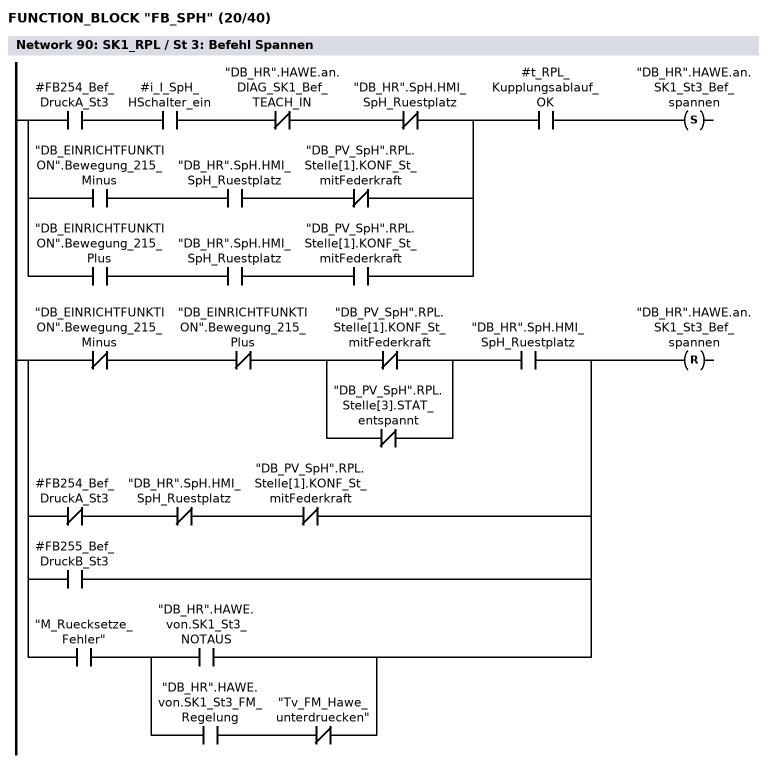

      U(    ;
      U     #FB254_Bef_DruckA_St3;
      U     #i_I_SpH_HSchalter_ein;
      UN    "DB_HR".HAWE.an.DIAG_SK1_Bef_TEACH_IN;
      UN    "DB_HR".SpH.HMI_SpH_Ruestplatz;
      O     ;
      U     "DB_EINRICHTFUNKTION".Bewegung_215_Minus;
      U     "DB_HR".SpH.HMI_SpH_Ruestplatz;
      UN    "DB_PV_SpH".RPL.Stelle[1].KONF_St_mitFederkraft;
      O     ;
      U     "DB_EINRICHTFUNKTION".Bewegung_215_Plus;
      U     "DB_HR".SpH.HMI_SpH_Ruestplatz;
      U     "DB_PV_SpH".RPL.Stelle[1].KONF_St_mitFederkraft;
      )     ;
      U     #t_RPL_Kupplungsablauf_OK;
      S     "DB_HR".HAWE.an.SK1_St3_Bef_spannen;

      U(    ;
      UN    "DB_EINRICHTFUNKTION".Bewegung_215_Minus;
      UN    "DB_EINRICHTFUNKTION".Bewegung_215_Plus;
      U(    ;
      ON    "DB_PV_SpH".RPL.Stelle[1].KONF_St_mitFederkraft;
      ON    "DB_PV_SpH".RPL.Stelle[3].STAT_entspannt;
      )     ;
      U     "DB_HR".SpH.HMI_SpH_Ruestplatz;
      O     ;
      UN    #FB254_Bef_DruckA_St3;
      UN    "DB_HR".SpH.HMI_SpH_Ruestplatz;
      UN    "DB_PV_SpH".RPL.Stelle[1].KONF_St_mitFederkraft;
      O     #FB255_Bef_DruckB_St3;
      O     ;
      U     "M_Ruecksetze_Fehler";
      U(    ;
      O     "DB_HR".HAWE.von.SK1_St3_NOTAUS;
      O     ;
      U     "DB_HR".HAWE.von.SK1_St3_FM_Regelung;
      UN    "Tv_FM_Hawe_unterdruecken";
      )     ;
      )     ;
      R     "DB_HR".HAWE.an.SK1_St3_Bef_spannen;
      NOP   0;
NETWORK
TITLE =SK1_RPL / St 4: Befehl Spannen
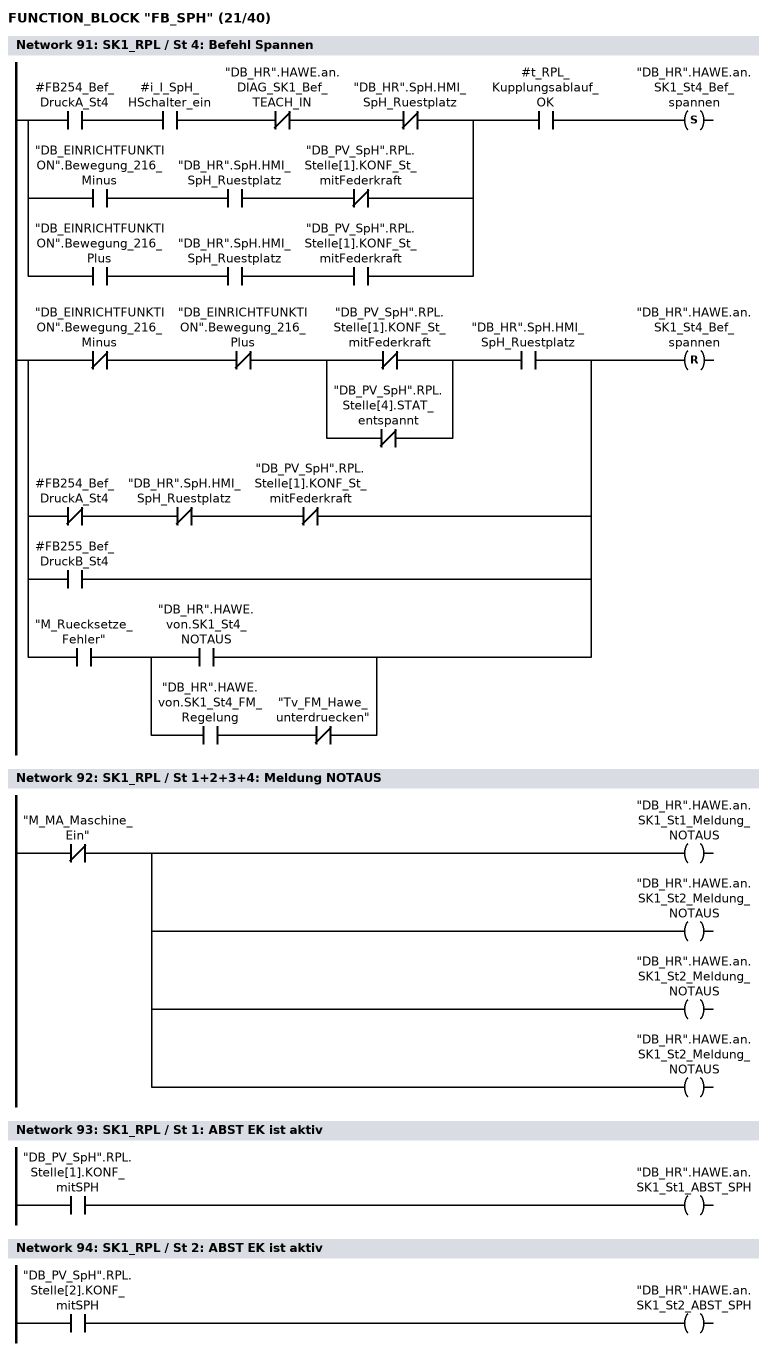

      U(    ;
      U     #FB254_Bef_DruckA_St4;
      U     #i_I_SpH_HSchalter_ein;
      UN    "DB_HR".HAWE.an.DIAG_SK1_Bef_TEACH_IN;
      UN    "DB_HR".SpH.HMI_SpH_Ruestplatz;
      O     ;
      U     "DB_EINRICHTFUNKTION".Bewegung_216_Minus;
      U     "DB_HR".SpH.HMI_SpH_Ruestplatz;
      UN    "DB_PV_SpH".RPL.Stelle[1].KONF_St_mitFederkraft;
      O     ;
      U     "DB_EINRICHTFUNKTION".Bewegung_216_Plus;
      U     "DB_HR".SpH.HMI_SpH_Ruestplatz;
      U     "DB_PV_SpH".RPL.Stelle[1].KONF_St_mitFederkraft;
      )     ;
      U     #t_RPL_Kupplungsablauf_OK;
      S     "DB_HR".HAWE.an.SK1_St4_Bef_spannen;

      U(    ;
      UN    "DB_EINRICHTFUNKTION".Bewegung_216_Minus;
      UN    "DB_EINRICHTFUNKTION".Bewegung_216_Plus;
      U(    ;
      ON    "DB_PV_SpH".RPL.Stelle[1].KONF_St_mitFederkraft;
      ON    "DB_PV_SpH".RPL.Stelle[4].STAT_entspannt;
      )     ;
      U     "DB_HR".SpH.HMI_SpH_Ruestplatz;
      O     ;
      UN    #FB254_Bef_DruckA_St4;
      UN    "DB_HR".SpH.HMI_SpH_Ruestplatz;
      UN    "DB_PV_SpH".RPL.Stelle[1].KONF_St_mitFederkraft;
      O     #FB255_Bef_DruckB_St4;
      O     ;
      U     "M_Ruecksetze_Fehler";
      U(    ;
      O     "DB_HR".HAWE.von.SK1_St4_NOTAUS;
      O     ;
      U     "DB_HR".HAWE.von.SK1_St4_FM_Regelung;
      UN    "Tv_FM_Hawe_unterdruecken";
      )     ;
      )     ;
      R     "DB_HR".HAWE.an.SK1_St4_Bef_spannen;
      NOP   0;
NETWORK
TITLE =SK1_RPL / St 1+2+3+4: Meldung NOTAUS

      UN    "M_MA_Maschine_Ein";
      =     "DB_HR".HAWE.an.SK1_St1_Meldung_NOTAUS;
      =     "DB_HR".HAWE.an.SK1_St2_Meldung_NOTAUS;
      =     "DB_HR".HAWE.an.SK1_St2_Meldung_NOTAUS;
      =     "DB_HR".HAWE.an.SK1_St2_Meldung_NOTAUS;
NETWORK
TITLE =SK1_RPL / St 1: ABST EK ist aktiv

      U     "DB_PV_SpH".RPL.Stelle[1].KONF_mitSPH;
      =     "DB_HR".HAWE.an.SK1_St1_ABST_SPH;
NETWORK
TITLE =SK1_RPL / St 2: ABST EK ist aktiv

      U     "DB_PV_SpH".RPL.Stelle[2].KONF_mitSPH;
      =     "DB_HR".HAWE.an.SK1_St2_ABST_SPH;
NETWORK
TITLE =SK1_RPL / St 3: ABST EK ist aktiv
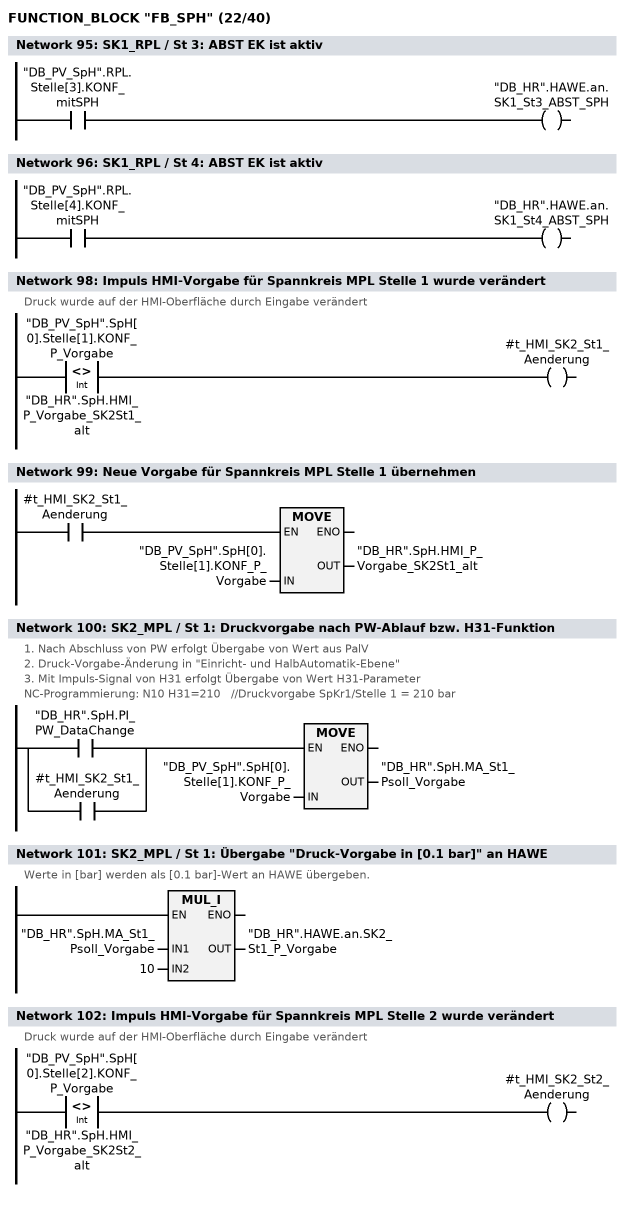

      U     "DB_PV_SpH".RPL.Stelle[3].KONF_mitSPH;
      =     "DB_HR".HAWE.an.SK1_St3_ABST_SPH;
NETWORK
TITLE =SK1_RPL / St 4: ABST EK ist aktiv

      U     "DB_PV_SpH".RPL.Stelle[4].KONF_mitSPH;
      =     "DB_HR".HAWE.an.SK1_St4_ABST_SPH;
NETWORK
TITLE =-------------- Maschinenplatz-Datenübergabe an HAWE ------------



NETWORK
TITLE =Impuls HMI-Vorgabe für Spannkreis MPL Stelle 1 wurde verändert
//Druck wurde auf der HMI-Oberfläche durch Eingabe verändert
      L     "DB_PV_SpH".SpH[0].Stelle[1].KONF_P_Vorgabe;
      L     "DB_HR".SpH.HMI_P_Vorgabe_SK2St1_alt;
      <>I   ;
      =     #t_HMI_SK2_St1_Aenderung;
NETWORK
TITLE =Neue Vorgabe für Spannkreis MPL Stelle 1 übernehmen

      U     #t_HMI_SK2_St1_Aenderung;
      SPBNB _00a;
      L     "DB_PV_SpH".SpH[0].Stelle[1].KONF_P_Vorgabe;
      T     "DB_HR".SpH.HMI_P_Vorgabe_SK2St1_alt;
_00a: NOP   0;
NETWORK
TITLE =SK2_MPL / St 1: Druckvorgabe nach PW-Ablauf bzw. H31-Funktion
//1. Nach Abschluss von PW erfolgt Übergabe von Wert aus PalV
//2. Druck-Vorgabe-Änderung in "Einricht- und HalbAutomatik-Ebene"
//3. Mit Impuls-Signal von H31 erfolgt Übergabe von Wert H31-Parameter
//   NC-Programmierung: N10 H31=210   //Druckvorgabe SpKr1/Stelle 1 = 210 bar
      U(    ;
      O     "DB_HR".SpH.PI_PW_DataChange;
      O     #t_HMI_SK2_St1_Aenderung;
      )     ;
      SPBNB _00b;
      L     "DB_PV_SpH".SpH[0].Stelle[1].KONF_P_Vorgabe;
      T     "DB_HR".SpH.MA_St1_Psoll_Vorgabe;
_00b: NOP   0;
NETWORK
TITLE =SK2_MPL / St 1: Übergabe "Druck-Vorgabe in [0.1 bar]" an HAWE
//Werte in [bar] werden als [0.1 bar]-Wert an HAWE übergeben.
      L     "DB_HR".SpH.MA_St1_Psoll_Vorgabe;
      L     10;
      *I    ;
      T     "DB_HR".HAWE.an.SK2_St1_P_Vorgabe;
NETWORK
TITLE =Impuls HMI-Vorgabe für Spannkreis MPL Stelle 2 wurde verändert
//Druck wurde auf der HMI-Oberfläche durch Eingabe verändert
      L     "DB_PV_SpH".SpH[0].Stelle[2].KONF_P_Vorgabe;
      L     "DB_HR".SpH.HMI_P_Vorgabe_SK2St2_alt;
      <>I   ;
      =     #t_HMI_SK2_St2_Aenderung;
NETWORK
TITLE =Neue Vorgabe für Spannkreis MPL Stelle 2 übernehmen
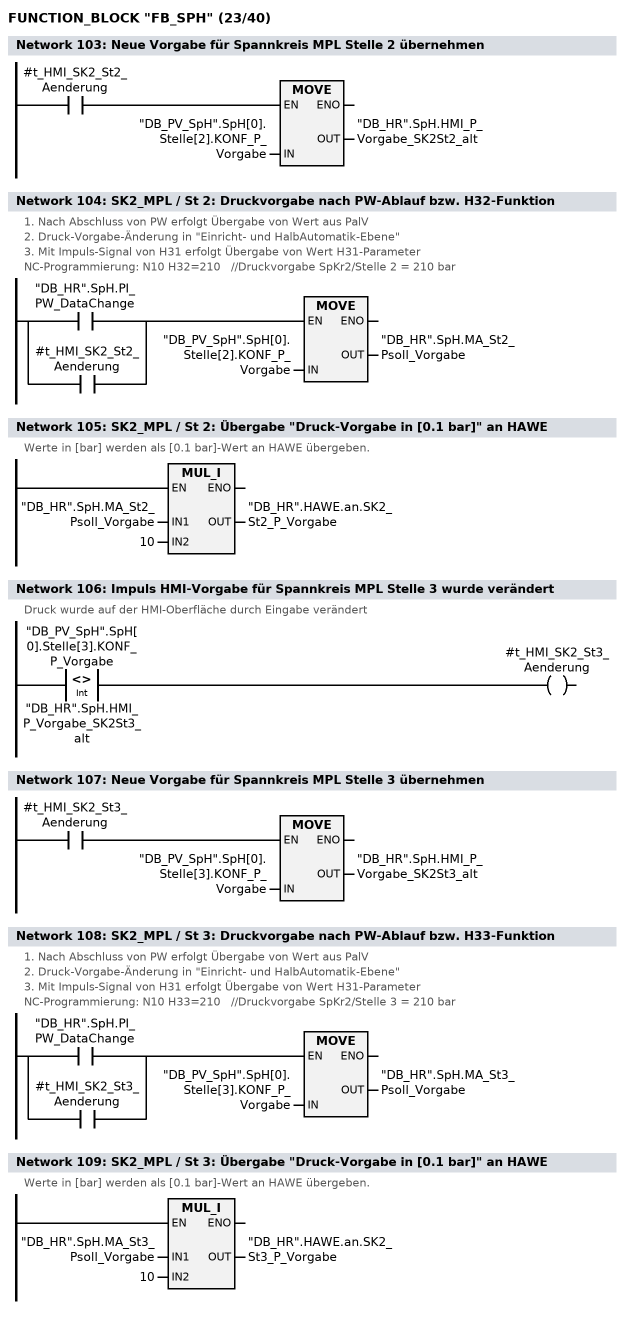

      U     #t_HMI_SK2_St2_Aenderung;
      SPBNB _00c;
      L     "DB_PV_SpH".SpH[0].Stelle[2].KONF_P_Vorgabe;
      T     "DB_HR".SpH.HMI_P_Vorgabe_SK2St2_alt;
_00c: NOP   0;
NETWORK
TITLE =SK2_MPL / St 2: Druckvorgabe nach PW-Ablauf bzw. H32-Funktion
//1. Nach Abschluss von PW erfolgt Übergabe von Wert aus PalV
//2. Druck-Vorgabe-Änderung in "Einricht- und HalbAutomatik-Ebene"
//3. Mit Impuls-Signal von H31 erfolgt Übergabe von Wert H31-Parameter
//   NC-Programmierung: N10 H32=210   //Druckvorgabe SpKr2/Stelle 2 = 210 bar
      U(    ;
      O     "DB_HR".SpH.PI_PW_DataChange;
      O     #t_HMI_SK2_St2_Aenderung;
      )     ;
      SPBNB _00d;
      L     "DB_PV_SpH".SpH[0].Stelle[2].KONF_P_Vorgabe;
      T     "DB_HR".SpH.MA_St2_Psoll_Vorgabe;
_00d: NOP   0;
NETWORK
TITLE =SK2_MPL / St 2: Übergabe "Druck-Vorgabe in [0.1 bar]" an HAWE
//Werte in [bar] werden als [0.1 bar]-Wert an HAWE übergeben.
      L     "DB_HR".SpH.MA_St2_Psoll_Vorgabe;
      L     10;
      *I    ;
      T     "DB_HR".HAWE.an.SK2_St2_P_Vorgabe;
NETWORK
TITLE =Impuls HMI-Vorgabe für Spannkreis MPL Stelle 3 wurde verändert
//Druck wurde auf der HMI-Oberfläche durch Eingabe verändert
      L     "DB_PV_SpH".SpH[0].Stelle[3].KONF_P_Vorgabe;
      L     "DB_HR".SpH.HMI_P_Vorgabe_SK2St3_alt;
      <>I   ;
      =     #t_HMI_SK2_St3_Aenderung;
NETWORK
TITLE =Neue Vorgabe für Spannkreis MPL Stelle 3 übernehmen

      U     #t_HMI_SK2_St3_Aenderung;
      SPBNB _00e;
      L     "DB_PV_SpH".SpH[0].Stelle[3].KONF_P_Vorgabe;
      T     "DB_HR".SpH.HMI_P_Vorgabe_SK2St3_alt;
_00e: NOP   0;
NETWORK
TITLE =SK2_MPL / St 3: Druckvorgabe nach PW-Ablauf bzw. H33-Funktion
//1. Nach Abschluss von PW erfolgt Übergabe von Wert aus PalV
//2. Druck-Vorgabe-Änderung in "Einricht- und HalbAutomatik-Ebene"
//3. Mit Impuls-Signal von H31 erfolgt Übergabe von Wert H31-Parameter
//   NC-Programmierung: N10 H33=210   //Druckvorgabe SpKr2/Stelle 3 = 210 bar
      U(    ;
      O     "DB_HR".SpH.PI_PW_DataChange;
      O     #t_HMI_SK2_St3_Aenderung;
      )     ;
      SPBNB _00f;
      L     "DB_PV_SpH".SpH[0].Stelle[3].KONF_P_Vorgabe;
      T     "DB_HR".SpH.MA_St3_Psoll_Vorgabe;
_00f: NOP   0;
NETWORK
TITLE =SK2_MPL / St 3: Übergabe "Druck-Vorgabe in [0.1 bar]" an HAWE
//Werte in [bar] werden als [0.1 bar]-Wert an HAWE übergeben.
      L     "DB_HR".SpH.MA_St3_Psoll_Vorgabe;
      L     10;
      *I    ;
      T     "DB_HR".HAWE.an.SK2_St3_P_Vorgabe;
NETWORK
TITLE =Impuls HMI-Vorgabe für Spannkreis MPL Stelle 4 wurde verändert
//Druck wurde auf der HMI-Oberfläche durch Eingabe verändert
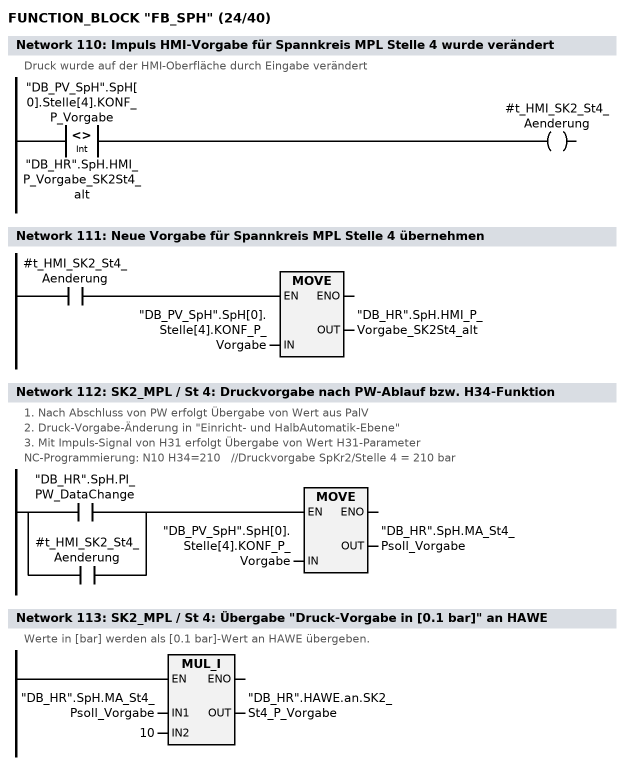
      L     "DB_PV_SpH".SpH[0].Stelle[4].KONF_P_Vorgabe;
      L     "DB_HR".SpH.HMI_P_Vorgabe_SK2St4_alt;
      <>I   ;
      =     #t_HMI_SK2_St4_Aenderung;
NETWORK
TITLE =Neue Vorgabe für Spannkreis MPL Stelle 4 übernehmen

      U     #t_HMI_SK2_St4_Aenderung;
      SPBNB _010;
      L     "DB_PV_SpH".SpH[0].Stelle[4].KONF_P_Vorgabe;
      T     "DB_HR".SpH.HMI_P_Vorgabe_SK2St4_alt;
_010: NOP   0;
NETWORK
TITLE =SK2_MPL / St 4: Druckvorgabe nach PW-Ablauf bzw. H34-Funktion
//1. Nach Abschluss von PW erfolgt Übergabe von Wert aus PalV
//2. Druck-Vorgabe-Änderung in "Einricht- und HalbAutomatik-Ebene"
//3. Mit Impuls-Signal von H31 erfolgt Übergabe von Wert H31-Parameter
//   NC-Programmierung: N10 H34=210   //Druckvorgabe SpKr2/Stelle 4 = 210 bar
      U(    ;
      O     "DB_HR".SpH.PI_PW_DataChange;
      O     #t_HMI_SK2_St4_Aenderung;
      )     ;
      SPBNB _011;
      L     "DB_PV_SpH".SpH[0].Stelle[4].KONF_P_Vorgabe;
      T     "DB_HR".SpH.MA_St4_Psoll_Vorgabe;
_011: NOP   0;
NETWORK
TITLE =SK2_MPL / St 4: Übergabe "Druck-Vorgabe in [0.1 bar]" an HAWE
//Werte in [bar] werden als [0.1 bar]-Wert an HAWE übergeben.
      L     "DB_HR".SpH.MA_St4_Psoll_Vorgabe;
      L     10;
      *I    ;
      T     "DB_HR".HAWE.an.SK2_St4_P_Vorgabe;
NETWORK
TITLE =H31-Funktion
//i_REAL_H_wert           := REAL-Wert der H-Funktion
//i_T_Ausgang_Entspannen  := Timer-Ausgang: Spannstelle entspannen
//i_HAWE_Druck_erreicht   := Meldung von HAWE "Druck erreicht"
//i_RESET_offene_Stelle_OK:= RESET Funktion "offene Spannstelle"
//                           z.B. PW-Ablauf aktiv
//i_Spannstelle_aktiv     := Spannstelle konfiguriert
//o_HFKT_quitpflichtig    := Merker für H-Funktion "Quittierungspflichtig"
//o_HFKT_Quittung         := Merker für H-Funktion "Quittierung"
//o_FM_falscher_Wert      := FM "Falscher Wert bei H-Eingabe"
//o_T_Start_Entspannen    := Timer-Start: Spannstelle entspannen
//o_T_Vorgabe_Entspannen  := Timer-Vorgabe: Spannstelle entspannen [s]
//o_kein_OVR_ist_0        := kein OVR=0 aktivieren
//                           a) Überwachung ist ausgeschaltet
//                           b) Spannstelle wurde geöffnet
//io_akt_Druckvorgabe     := Aktuelle Druckvorgabe (Sollwert in Maschine)
//io_M_H_FKT              := Merker für H-Funktion aktiv
//io_Bef_Entspannen       := Befehl an Hawe "Spannstelle entspannen"
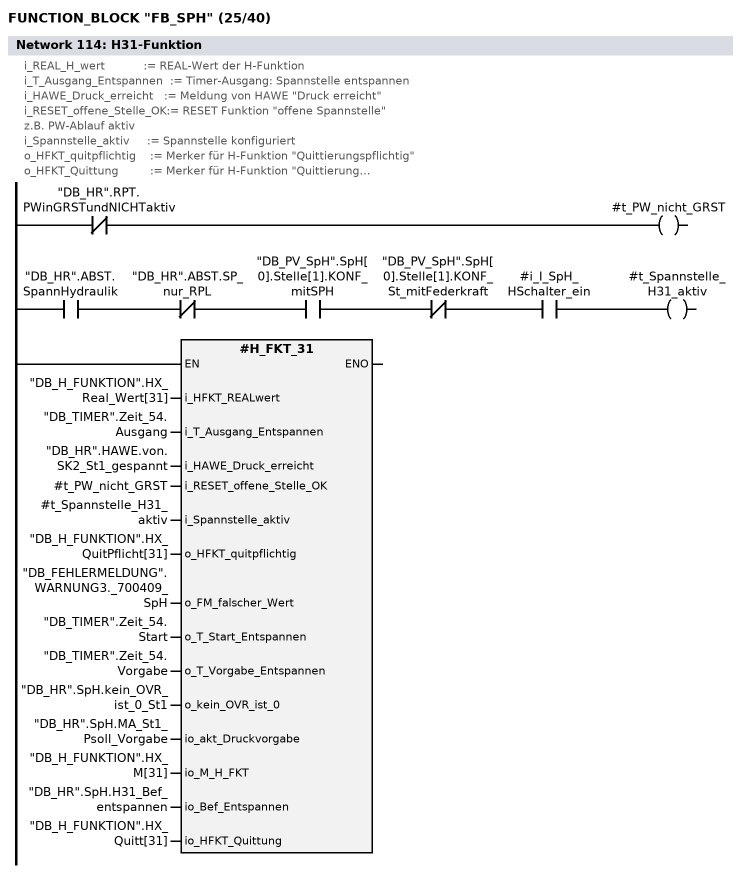
      UN    "DB_HR".RPT.PWinGRSTundNICHTaktiv;
      =     #t_PW_nicht_GRST;

      U     "DB_HR".ABST.SpannHydraulik;
      UN    "DB_HR".ABST.SP_nur_RPL;
      U     "DB_PV_SpH".SpH[0].Stelle[1].KONF_mitSPH;
      UN    "DB_PV_SpH".SpH[0].Stelle[1].KONF_St_mitFederkraft;
      U     #i_I_SpH_HSchalter_ein;
      =     #t_Spannstelle_H31_aktiv;

      CALL #H_FKT_31 (
           i_HFKT_REALwert          := "DB_H_FUNKTION".HX_Real_Wert[31],
           i_T_Ausgang_Entspannen   := "DB_TIMER".Zeit_54.Ausgang,
           i_HAWE_Druck_erreicht    := "DB_HR".HAWE.von.SK2_St1_gespannt,
           i_RESET_offene_Stelle_OK := #t_PW_nicht_GRST,
           i_Spannstelle_aktiv      := #t_Spannstelle_H31_aktiv,
           o_HFKT_quitpflichtig     := "DB_H_FUNKTION".HX_QuitPflicht[31],
           o_FM_falscher_Wert       := "DB_FEHLERMELDUNG".WARNUNG3._700409_SpH,
           o_T_Start_Entspannen     := "DB_TIMER".Zeit_54.Start,
           o_T_Vorgabe_Entspannen   := "DB_TIMER".Zeit_54.Vorgabe,
           o_kein_OVR_ist_0         := "DB_HR".SpH.kein_OVR_ist_0_St1,
           io_akt_Druckvorgabe      := "DB_HR".SpH.MA_St1_Psoll_Vorgabe,
           io_M_H_FKT               := "DB_H_FUNKTION".HX_M[31],
           io_Bef_Entspannen        := "DB_HR".SpH.H31_Bef_entspannen,
           io_HFKT_Quittung         := "DB_H_FUNKTION".HX_Quitt[31]);

NETWORK
TITLE =H32-Funktion
//i_REAL_H_wert           := REAL-Wert der H-Funktion
//i_T_Ausgang_Entspannen  := Timer-Ausgang: Spannstelle entspannen
//i_HAWE_Druck_erreicht   := Meldung von HAWE "Druck erreicht"
//i_RESET_offene_Stelle_OK:= RESET Funktion "offene Spannstelle"
//                           z.B. PW-Ablauf aktiv
//i_Spannstelle_aktiv     := Spannstelle konfiguriert
//o_HFKT_quitpflichtig    := Merker für H-Funktion "Quittierungspflichtig"
//o_HFKT_Quittung         := Merker für H-Funktion "Quittierung"
//o_FM_falscher_Wert      := FM "Falscher Wert bei H-Eingabe"
//o_T_Start_Entspannen    := Timer-Start: Spannstelle entspannen
//o_T_Vorgabe_Entspannen  := Timer-Vorgabe: Spannstelle entspannen [s]
//o_kein_OVR_ist_0        := kein OVR=0 aktivieren
//                           a) Überwachung ist ausgeschaltet
//                           b) Spannstelle wurde geöffnet
//io_akt_Druckvorgabe     := Aktuelle Druckvorgabe (Sollwert in Maschine)
//io_M_H_FKT              := Merker für H-Funktion aktiv
//io_Bef_Entspannen       := Befehl an Hawe "Spannstelle entspannen"
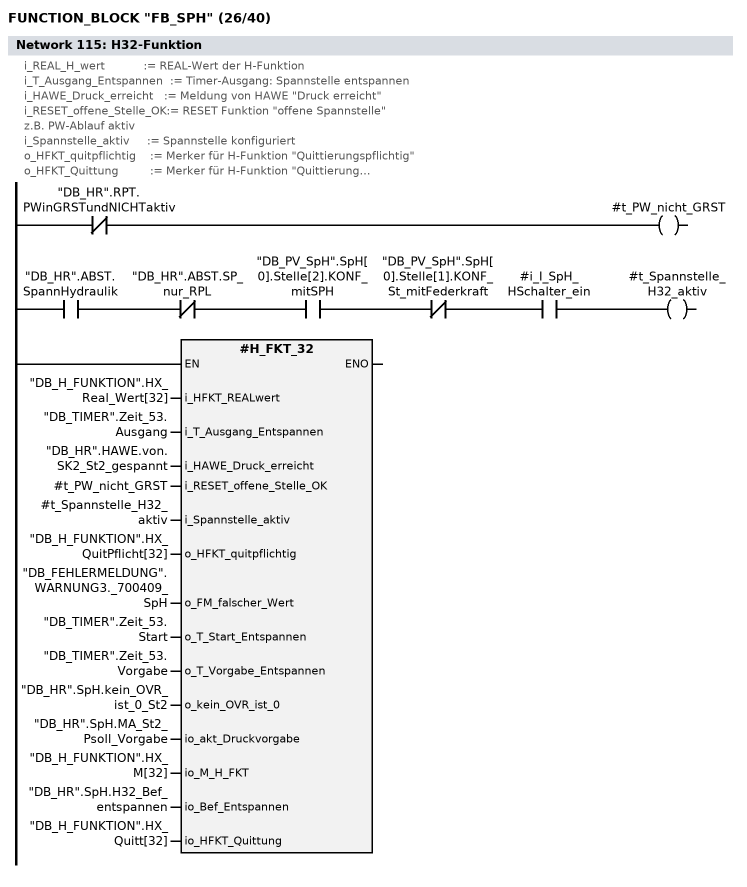
      UN    "DB_HR".RPT.PWinGRSTundNICHTaktiv;
      =     #t_PW_nicht_GRST;

      U     "DB_HR".ABST.SpannHydraulik;
      UN    "DB_HR".ABST.SP_nur_RPL;
      U     "DB_PV_SpH".SpH[0].Stelle[2].KONF_mitSPH;
      UN    "DB_PV_SpH".SpH[0].Stelle[1].KONF_St_mitFederkraft;
      U     #i_I_SpH_HSchalter_ein;
      =     #t_Spannstelle_H32_aktiv;

      CALL #H_FKT_32 (
           i_HFKT_REALwert          := "DB_H_FUNKTION".HX_Real_Wert[32],
           i_T_Ausgang_Entspannen   := "DB_TIMER".Zeit_53.Ausgang,
           i_HAWE_Druck_erreicht    := "DB_HR".HAWE.von.SK2_St2_gespannt,
           i_RESET_offene_Stelle_OK := #t_PW_nicht_GRST,
           i_Spannstelle_aktiv      := #t_Spannstelle_H32_aktiv,
           o_HFKT_quitpflichtig     := "DB_H_FUNKTION".HX_QuitPflicht[32],
           o_FM_falscher_Wert       := "DB_FEHLERMELDUNG".WARNUNG3._700409_SpH,
           o_T_Start_Entspannen     := "DB_TIMER".Zeit_53.Start,
           o_T_Vorgabe_Entspannen   := "DB_TIMER".Zeit_53.Vorgabe,
           o_kein_OVR_ist_0         := "DB_HR".SpH.kein_OVR_ist_0_St2,
           io_akt_Druckvorgabe      := "DB_HR".SpH.MA_St2_Psoll_Vorgabe,
           io_M_H_FKT               := "DB_H_FUNKTION".HX_M[32],
           io_Bef_Entspannen        := "DB_HR".SpH.H32_Bef_entspannen,
           io_HFKT_Quittung         := "DB_H_FUNKTION".HX_Quitt[32]);

NETWORK
TITLE =H33-Funktion
//i_REAL_H_wert           := REAL-Wert der H-Funktion
//i_T_Ausgang_Entspannen  := Timer-Ausgang: Spannstelle entspannen
//i_HAWE_Druck_erreicht   := Meldung von HAWE "Druck erreicht"
//i_RESET_offene_Stelle_OK:= RESET Funktion "offene Spannstelle"
//                           z.B. PW-Ablauf aktiv
//i_Spannstelle_aktiv     := Spannstelle konfiguriert
//o_HFKT_quitpflichtig    := Merker für H-Funktion "Quittierungspflichtig"
//o_HFKT_Quittung         := Merker für H-Funktion "Quittierung"
//o_FM_falscher_Wert      := FM "Falscher Wert bei H-Eingabe"
//o_T_Start_Entspannen    := Timer-Start: Spannstelle entspannen
//o_T_Vorgabe_Entspannen  := Timer-Vorgabe: Spannstelle entspannen [s]
//o_kein_OVR_ist_0        := kein OVR=0 aktivieren
//                           a) Überwachung ist ausgeschaltet
//                           b) Spannstelle wurde geöffnet
//io_akt_Druckvorgabe     := Aktuelle Druckvorgabe (Sollwert in Maschine)
//io_M_H_FKT              := Merker für H-Funktion aktiv
//io_Bef_Entspannen       := Befehl an Hawe "Spannstelle entspannen"
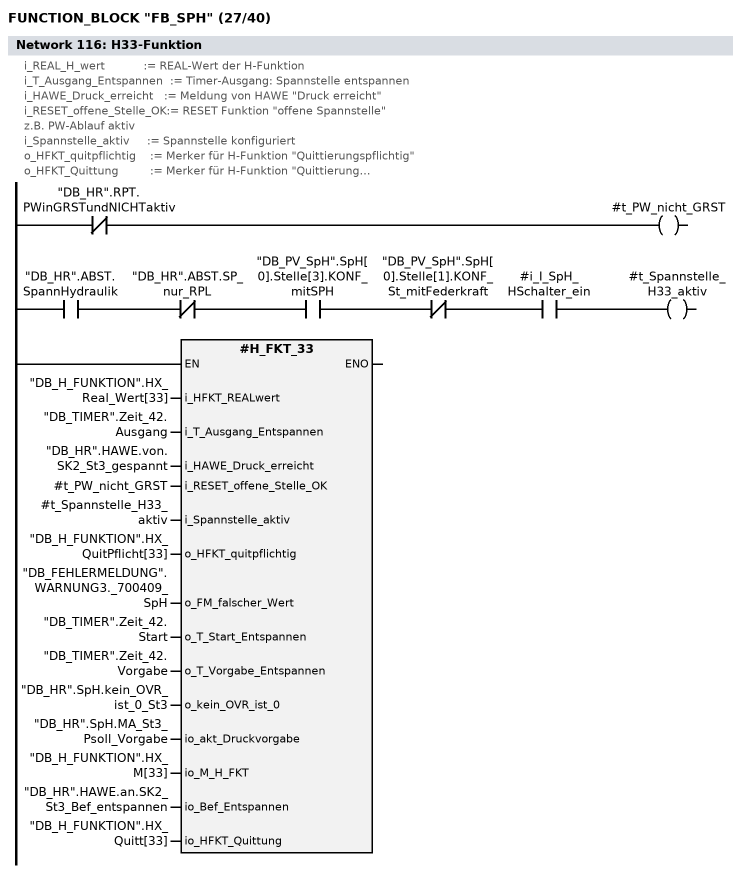
      UN    "DB_HR".RPT.PWinGRSTundNICHTaktiv;
      =     #t_PW_nicht_GRST;

      U     "DB_HR".ABST.SpannHydraulik;
      UN    "DB_HR".ABST.SP_nur_RPL;
      U     "DB_PV_SpH".SpH[0].Stelle[3].KONF_mitSPH;
      UN    "DB_PV_SpH".SpH[0].Stelle[1].KONF_St_mitFederkraft;
      U     #i_I_SpH_HSchalter_ein;
      =     #t_Spannstelle_H33_aktiv;


      CALL #H_FKT_33 (
           i_HFKT_REALwert          := "DB_H_FUNKTION".HX_Real_Wert[33],
           i_T_Ausgang_Entspannen   := "DB_TIMER".Zeit_42.Ausgang,
           i_HAWE_Druck_erreicht    := "DB_HR".HAWE.von.SK2_St3_gespannt,
           i_RESET_offene_Stelle_OK := #t_PW_nicht_GRST,
           i_Spannstelle_aktiv      := #t_Spannstelle_H33_aktiv,
           o_HFKT_quitpflichtig     := "DB_H_FUNKTION".HX_QuitPflicht[33],
           o_FM_falscher_Wert       := "DB_FEHLERMELDUNG".WARNUNG3._700409_SpH,
           o_T_Start_Entspannen     := "DB_TIMER".Zeit_42.Start,
           o_T_Vorgabe_Entspannen   := "DB_TIMER".Zeit_42.Vorgabe,
           o_kein_OVR_ist_0         := "DB_HR".SpH.kein_OVR_ist_0_St3,
           io_akt_Druckvorgabe      := "DB_HR".SpH.MA_St3_Psoll_Vorgabe,
           io_M_H_FKT               := "DB_H_FUNKTION".HX_M[33],
           io_Bef_Entspannen        := "DB_HR".HAWE.an.SK2_St3_Bef_entspannen,
           io_HFKT_Quittung         := "DB_H_FUNKTION".HX_Quitt[33]);

NETWORK
TITLE =H34-Funktion
//i_REAL_H_wert           := REAL-Wert der H-Funktion
//i_T_Ausgang_Entspannen  := Timer-Ausgang: Spannstelle entspannen
//i_HAWE_Druck_erreicht   := Meldung von HAWE "Druck erreicht"
//i_RESET_offene_Stelle_OK:= RESET Funktion "offene Spannstelle"
//                           z.B. PW-Ablauf aktiv
//i_Spannstelle_aktiv     := Spannstelle konfiguriert
//o_HFKT_quitpflichtig    := Merker für H-Funktion "Quittierungspflichtig"
//o_HFKT_Quittung         := Merker für H-Funktion "Quittierung"
//o_FM_falscher_Wert      := FM "Falscher Wert bei H-Eingabe"
//o_T_Start_Entspannen    := Timer-Start: Spannstelle entspannen
//o_T_Vorgabe_Entspannen  := Timer-Vorgabe: Spannstelle entspannen [s]
//o_kein_OVR_ist_0        := kein OVR=0 aktivieren
//                           a) Überwachung ist ausgeschaltet
//                           b) Spannstelle wurde geöffnet
//io_akt_Druckvorgabe     := Aktuelle Druckvorgabe (Sollwert in Maschine)
//io_M_H_FKT              := Merker für H-Funktion aktiv
//io_Bef_Entspannen       := Befehl an Hawe "Spannstelle entspannen"
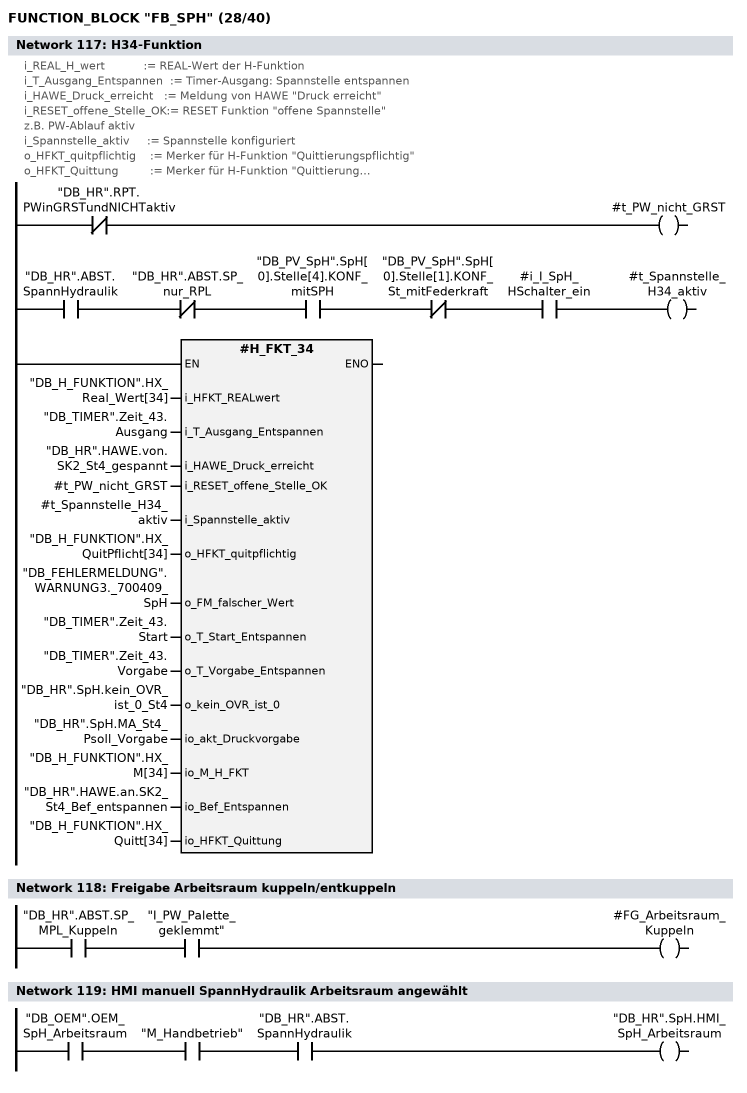
      UN    "DB_HR".RPT.PWinGRSTundNICHTaktiv;
      =     #t_PW_nicht_GRST;

      U     "DB_HR".ABST.SpannHydraulik;
      UN    "DB_HR".ABST.SP_nur_RPL;
      U     "DB_PV_SpH".SpH[0].Stelle[4].KONF_mitSPH;
      UN    "DB_PV_SpH".SpH[0].Stelle[1].KONF_St_mitFederkraft;
      U     #i_I_SpH_HSchalter_ein;
      =     #t_Spannstelle_H34_aktiv;

      CALL #H_FKT_34 (
           i_HFKT_REALwert          := "DB_H_FUNKTION".HX_Real_Wert[34],
           i_T_Ausgang_Entspannen   := "DB_TIMER".Zeit_43.Ausgang,
           i_HAWE_Druck_erreicht    := "DB_HR".HAWE.von.SK2_St4_gespannt,
           i_RESET_offene_Stelle_OK := #t_PW_nicht_GRST,
           i_Spannstelle_aktiv      := #t_Spannstelle_H34_aktiv,
           o_HFKT_quitpflichtig     := "DB_H_FUNKTION".HX_QuitPflicht[34],
           o_FM_falscher_Wert       := "DB_FEHLERMELDUNG".WARNUNG3._700409_SpH,
           o_T_Start_Entspannen     := "DB_TIMER".Zeit_43.Start,
           o_T_Vorgabe_Entspannen   := "DB_TIMER".Zeit_43.Vorgabe,
           o_kein_OVR_ist_0         := "DB_HR".SpH.kein_OVR_ist_0_St4,
           io_akt_Druckvorgabe      := "DB_HR".SpH.MA_St4_Psoll_Vorgabe,
           io_M_H_FKT               := "DB_H_FUNKTION".HX_M[34],
           io_Bef_Entspannen        := "DB_HR".HAWE.an.SK2_St4_Bef_entspannen,
           io_HFKT_Quittung         := "DB_H_FUNKTION".HX_Quitt[34]);
NETWORK
TITLE =Freigabe Arbeitsraum kuppeln/entkuppeln

      U     "DB_HR".ABST.SP_MPL_Kuppeln;
      U     "I_PW_Palette_geklemmt";
      =     #FG_Arbeitsraum_Kuppeln;
NETWORK
TITLE =HMI manuell SpannHydraulik Arbeitsraum angewählt

      U     "DB_OEM".OEM_SpH_Arbeitsraum;
      U     "M_Handbetrieb";
      U     "DB_HR".ABST.SpannHydraulik;
      =     "DB_HR".SpH.HMI_SpH_Arbeitsraum;
NETWORK
TITLE =HMI-Manuell: Maschinenraum Stelle 1
//HMI: Manuell / [SK5] Hand-Fkt SpannHydr.   Bild-Nr: 37
//                                           Bewegungs-Nr: 219
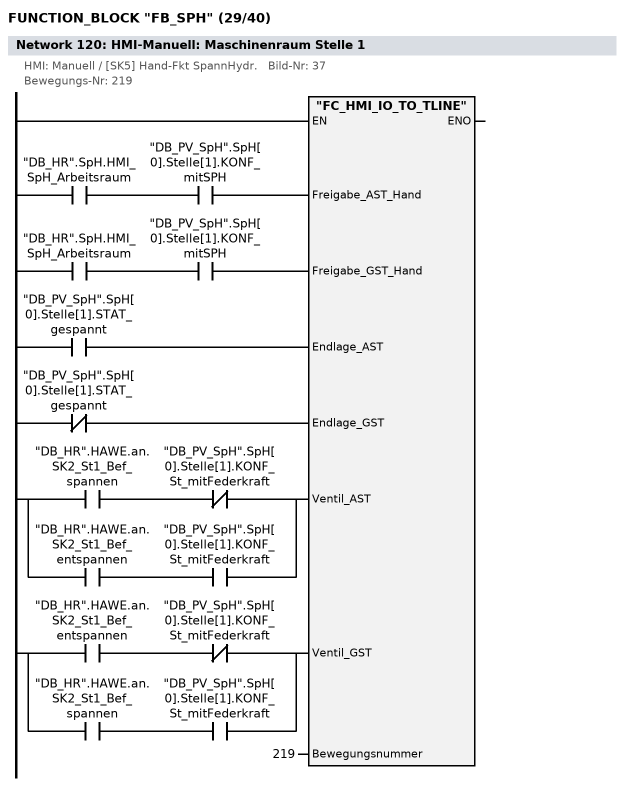
      U     "DB_HR".SpH.HMI_SpH_Arbeitsraum;
      U     "DB_PV_SpH".SpH[0].Stelle[1].KONF_mitSPH;
      =     L     18.0;
      BLD   103;
      U     "DB_HR".SpH.HMI_SpH_Arbeitsraum;
      U     "DB_PV_SpH".SpH[0].Stelle[1].KONF_mitSPH;
      =     L     18.1;
      BLD   103;
      U     "DB_PV_SpH".SpH[0].Stelle[1].STAT_gespannt;
      =     L     18.2;
      BLD   103;
      UN    "DB_PV_SpH".SpH[0].Stelle[1].STAT_gespannt;
      =     L     18.3;
      BLD   103;
      U(    ;
      U     "DB_HR".HAWE.an.SK2_St1_Bef_spannen;
      UN    "DB_PV_SpH".SpH[0].Stelle[1].KONF_St_mitFederkraft;
      O     ;
      U     "DB_HR".HAWE.an.SK2_St1_Bef_entspannen;
      U     "DB_PV_SpH".SpH[0].Stelle[1].KONF_St_mitFederkraft;
      )     ;
      =     L     18.4;
      BLD   103;
      U(    ;
      U     "DB_HR".HAWE.an.SK2_St1_Bef_entspannen;
      UN    "DB_PV_SpH".SpH[0].Stelle[1].KONF_St_mitFederkraft;
      O     ;
      U     "DB_HR".HAWE.an.SK2_St1_Bef_spannen;
      U     "DB_PV_SpH".SpH[0].Stelle[1].KONF_St_mitFederkraft;
      )     ;
      =     L     18.5;
      BLD   103;
      CALL "FC_HMI_IO_TO_TLINE" (
           Freigabe_AST_Hand        := L     18.0,
           Freigabe_GST_Hand        := L     18.1,
           Endlage_AST              := L     18.2,
           Endlage_GST              := L     18.3,
           Ventil_AST               := L     18.4,
           Ventil_GST               := L     18.5,
           Bewegungsnummer          := 219);
      NOP   0;
NETWORK
TITLE =HMI-Manuell: Maschinenraum Stelle 2
//HMI: Manuell / [SK5] Hand-Fkt SpannHydr.   Bild-Nr: 37
//                                           Bewegungs-Nr: 220
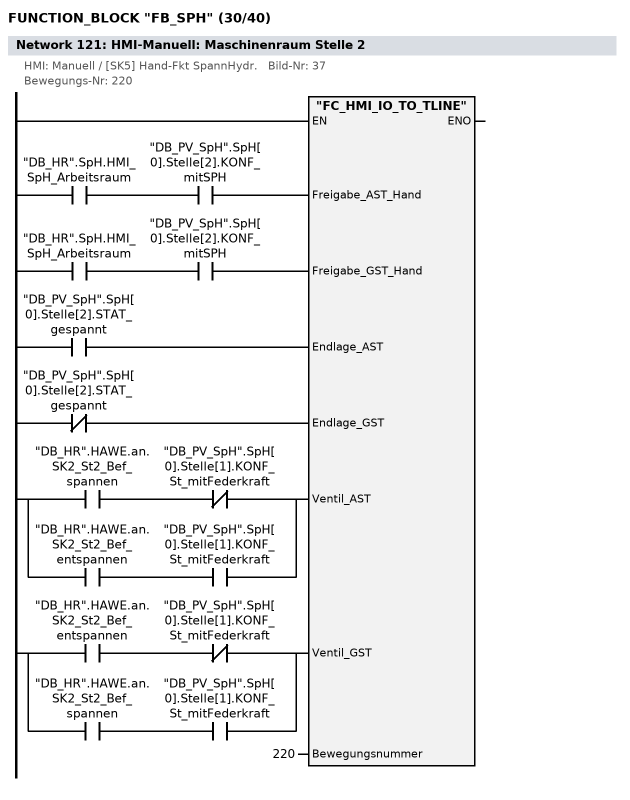
      U     "DB_HR".SpH.HMI_SpH_Arbeitsraum;
      U     "DB_PV_SpH".SpH[0].Stelle[2].KONF_mitSPH;
      =     L     18.0;
      BLD   103;
      U     "DB_HR".SpH.HMI_SpH_Arbeitsraum;
      U     "DB_PV_SpH".SpH[0].Stelle[2].KONF_mitSPH;
      =     L     18.1;
      BLD   103;
      U     "DB_PV_SpH".SpH[0].Stelle[2].STAT_gespannt;
      =     L     18.2;
      BLD   103;
      UN    "DB_PV_SpH".SpH[0].Stelle[2].STAT_gespannt;
      =     L     18.3;
      BLD   103;
      U(    ;
      U     "DB_HR".HAWE.an.SK2_St2_Bef_spannen;
      UN    "DB_PV_SpH".SpH[0].Stelle[1].KONF_St_mitFederkraft;
      O     ;
      U     "DB_HR".HAWE.an.SK2_St2_Bef_entspannen;
      U     "DB_PV_SpH".SpH[0].Stelle[1].KONF_St_mitFederkraft;
      )     ;
      =     L     18.4;
      BLD   103;
      U(    ;
      U     "DB_HR".HAWE.an.SK2_St2_Bef_entspannen;
      UN    "DB_PV_SpH".SpH[0].Stelle[1].KONF_St_mitFederkraft;
      O     ;
      U     "DB_HR".HAWE.an.SK2_St2_Bef_spannen;
      U     "DB_PV_SpH".SpH[0].Stelle[1].KONF_St_mitFederkraft;
      )     ;
      =     L     18.5;
      BLD   103;
      CALL "FC_HMI_IO_TO_TLINE" (
           Freigabe_AST_Hand        := L     18.0,
           Freigabe_GST_Hand        := L     18.1,
           Endlage_AST              := L     18.2,
           Endlage_GST              := L     18.3,
           Ventil_AST               := L     18.4,
           Ventil_GST               := L     18.5,
           Bewegungsnummer          := 220);
      NOP   0;
NETWORK
TITLE =HMI-Manuell: Maschinenraum Stelle 3
//HMI: Manuell / [SK5] Hand-Fkt SpannHydr.   Bild-Nr: 37
//                                           Bewegungs-Nr: 221
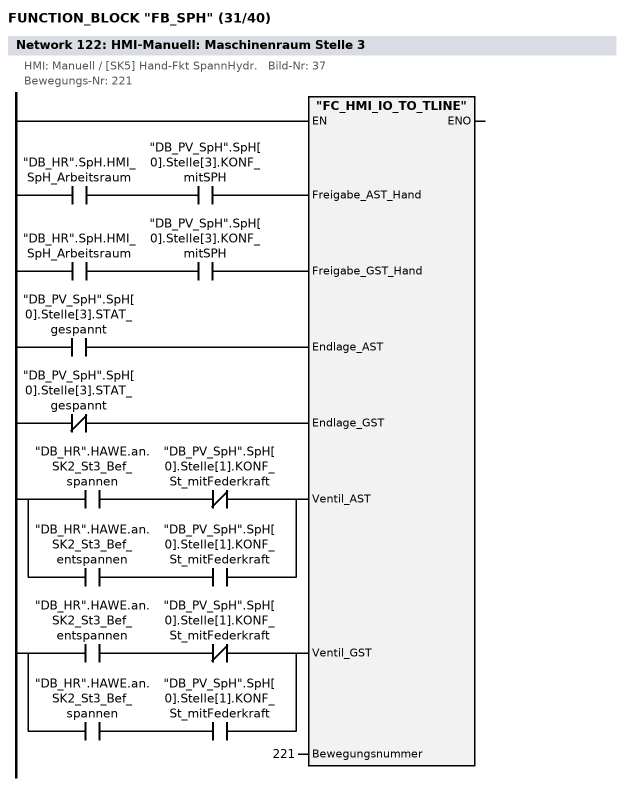
      U     "DB_HR".SpH.HMI_SpH_Arbeitsraum;
      U     "DB_PV_SpH".SpH[0].Stelle[3].KONF_mitSPH;
      =     L     18.0;
      BLD   103;
      U     "DB_HR".SpH.HMI_SpH_Arbeitsraum;
      U     "DB_PV_SpH".SpH[0].Stelle[3].KONF_mitSPH;
      =     L     18.1;
      BLD   103;
      U     "DB_PV_SpH".SpH[0].Stelle[3].STAT_gespannt;
      =     L     18.2;
      BLD   103;
      UN    "DB_PV_SpH".SpH[0].Stelle[3].STAT_gespannt;
      =     L     18.3;
      BLD   103;
      U(    ;
      U     "DB_HR".HAWE.an.SK2_St3_Bef_spannen;
      UN    "DB_PV_SpH".SpH[0].Stelle[1].KONF_St_mitFederkraft;
      O     ;
      U     "DB_HR".HAWE.an.SK2_St3_Bef_entspannen;
      U     "DB_PV_SpH".SpH[0].Stelle[1].KONF_St_mitFederkraft;
      )     ;
      =     L     18.4;
      BLD   103;
      U(    ;
      U     "DB_HR".HAWE.an.SK2_St3_Bef_entspannen;
      UN    "DB_PV_SpH".SpH[0].Stelle[1].KONF_St_mitFederkraft;
      O     ;
      U     "DB_HR".HAWE.an.SK2_St3_Bef_spannen;
      U     "DB_PV_SpH".SpH[0].Stelle[1].KONF_St_mitFederkraft;
      )     ;
      =     L     18.5;
      BLD   103;
      CALL "FC_HMI_IO_TO_TLINE" (
           Freigabe_AST_Hand        := L     18.0,
           Freigabe_GST_Hand        := L     18.1,
           Endlage_AST              := L     18.2,
           Endlage_GST              := L     18.3,
           Ventil_AST               := L     18.4,
           Ventil_GST               := L     18.5,
           Bewegungsnummer          := 221);
      NOP   0;
NETWORK
TITLE =HMI-Manuell: Maschinenraum Stelle 4
//HMI: Manuell / [SK5] Hand-Fkt SpannHydr.   Bild-Nr: 37
//                                           Bewegungs-Nr: 222
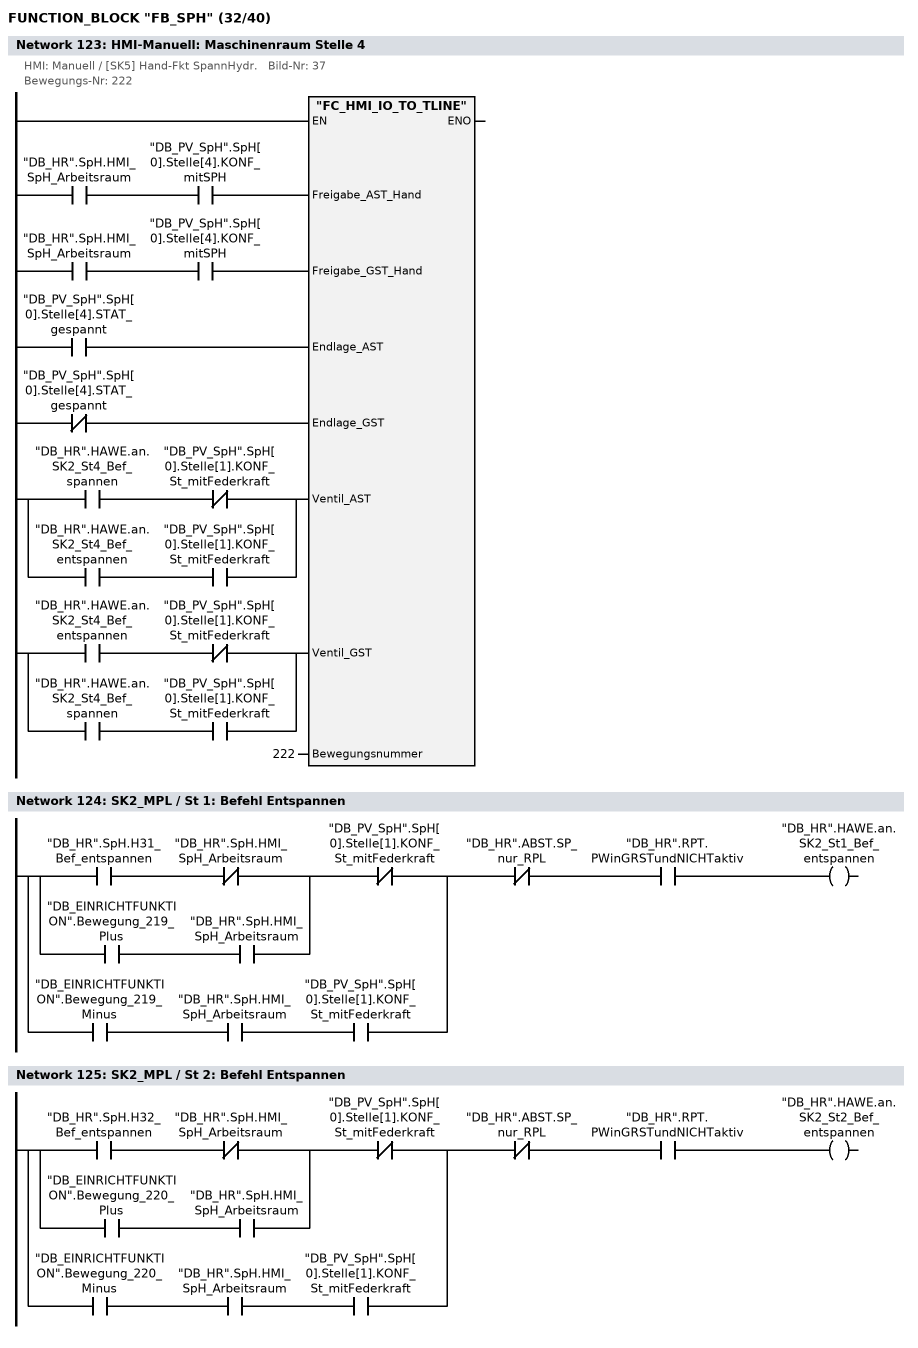
      U     "DB_HR".SpH.HMI_SpH_Arbeitsraum;
      U     "DB_PV_SpH".SpH[0].Stelle[4].KONF_mitSPH;
      =     L     18.0;
      BLD   103;
      U     "DB_HR".SpH.HMI_SpH_Arbeitsraum;
      U     "DB_PV_SpH".SpH[0].Stelle[4].KONF_mitSPH;
      =     L     18.1;
      BLD   103;
      U     "DB_PV_SpH".SpH[0].Stelle[4].STAT_gespannt;
      =     L     18.2;
      BLD   103;
      UN    "DB_PV_SpH".SpH[0].Stelle[4].STAT_gespannt;
      =     L     18.3;
      BLD   103;
      U(    ;
      U     "DB_HR".HAWE.an.SK2_St4_Bef_spannen;
      UN    "DB_PV_SpH".SpH[0].Stelle[1].KONF_St_mitFederkraft;
      O     ;
      U     "DB_HR".HAWE.an.SK2_St4_Bef_entspannen;
      U     "DB_PV_SpH".SpH[0].Stelle[1].KONF_St_mitFederkraft;
      )     ;
      =     L     18.4;
      BLD   103;
      U(    ;
      U     "DB_HR".HAWE.an.SK2_St4_Bef_entspannen;
      UN    "DB_PV_SpH".SpH[0].Stelle[1].KONF_St_mitFederkraft;
      O     ;
      U     "DB_HR".HAWE.an.SK2_St4_Bef_spannen;
      U     "DB_PV_SpH".SpH[0].Stelle[1].KONF_St_mitFederkraft;
      )     ;
      =     L     18.5;
      BLD   103;
      CALL "FC_HMI_IO_TO_TLINE" (
           Freigabe_AST_Hand        := L     18.0,
           Freigabe_GST_Hand        := L     18.1,
           Endlage_AST              := L     18.2,
           Endlage_GST              := L     18.3,
           Ventil_AST               := L     18.4,
           Ventil_GST               := L     18.5,
           Bewegungsnummer          := 222);
      NOP   0;
NETWORK
TITLE =SK2_MPL / St 1: Befehl Entspannen

      U(    ;
      U(    ;
      U     "DB_HR".SpH.H31_Bef_entspannen;
      UN    "DB_HR".SpH.HMI_SpH_Arbeitsraum;
      O     ;
      U     "DB_EINRICHTFUNKTION".Bewegung_219_Plus;
      U     "DB_HR".SpH.HMI_SpH_Arbeitsraum;
      )     ;
      UN    "DB_PV_SpH".SpH[0].Stelle[1].KONF_St_mitFederkraft;

      O     ;
      U     "DB_EINRICHTFUNKTION".Bewegung_219_Minus;
      U     "DB_HR".SpH.HMI_SpH_Arbeitsraum;
      U     "DB_PV_SpH".SpH[0].Stelle[1].KONF_St_mitFederkraft;
      )     ;
      UN    "DB_HR".ABST.SP_nur_RPL;
      U     "DB_HR".RPT.PWinGRSTundNICHTaktiv;
      =     "DB_HR".HAWE.an.SK2_St1_Bef_entspannen;
NETWORK
TITLE =SK2_MPL / St 2: Befehl Entspannen

      U(    ;
      U(    ;
      U     "DB_HR".SpH.H32_Bef_entspannen;
      UN    "DB_HR".SpH.HMI_SpH_Arbeitsraum;
      O     ;
      U     "DB_EINRICHTFUNKTION".Bewegung_220_Plus;
      U     "DB_HR".SpH.HMI_SpH_Arbeitsraum;
      )     ;
      UN    "DB_PV_SpH".SpH[0].Stelle[1].KONF_St_mitFederkraft;

      O     ;
      U     "DB_EINRICHTFUNKTION".Bewegung_220_Minus;
      U     "DB_HR".SpH.HMI_SpH_Arbeitsraum;
      U     "DB_PV_SpH".SpH[0].Stelle[1].KONF_St_mitFederkraft;
      )     ;
      UN    "DB_HR".ABST.SP_nur_RPL;
      U     "DB_HR".RPT.PWinGRSTundNICHTaktiv;
      =     "DB_HR".HAWE.an.SK2_St2_Bef_entspannen;
NETWORK
TITLE =SK2_MPL / St 3: Befehl Entspannen
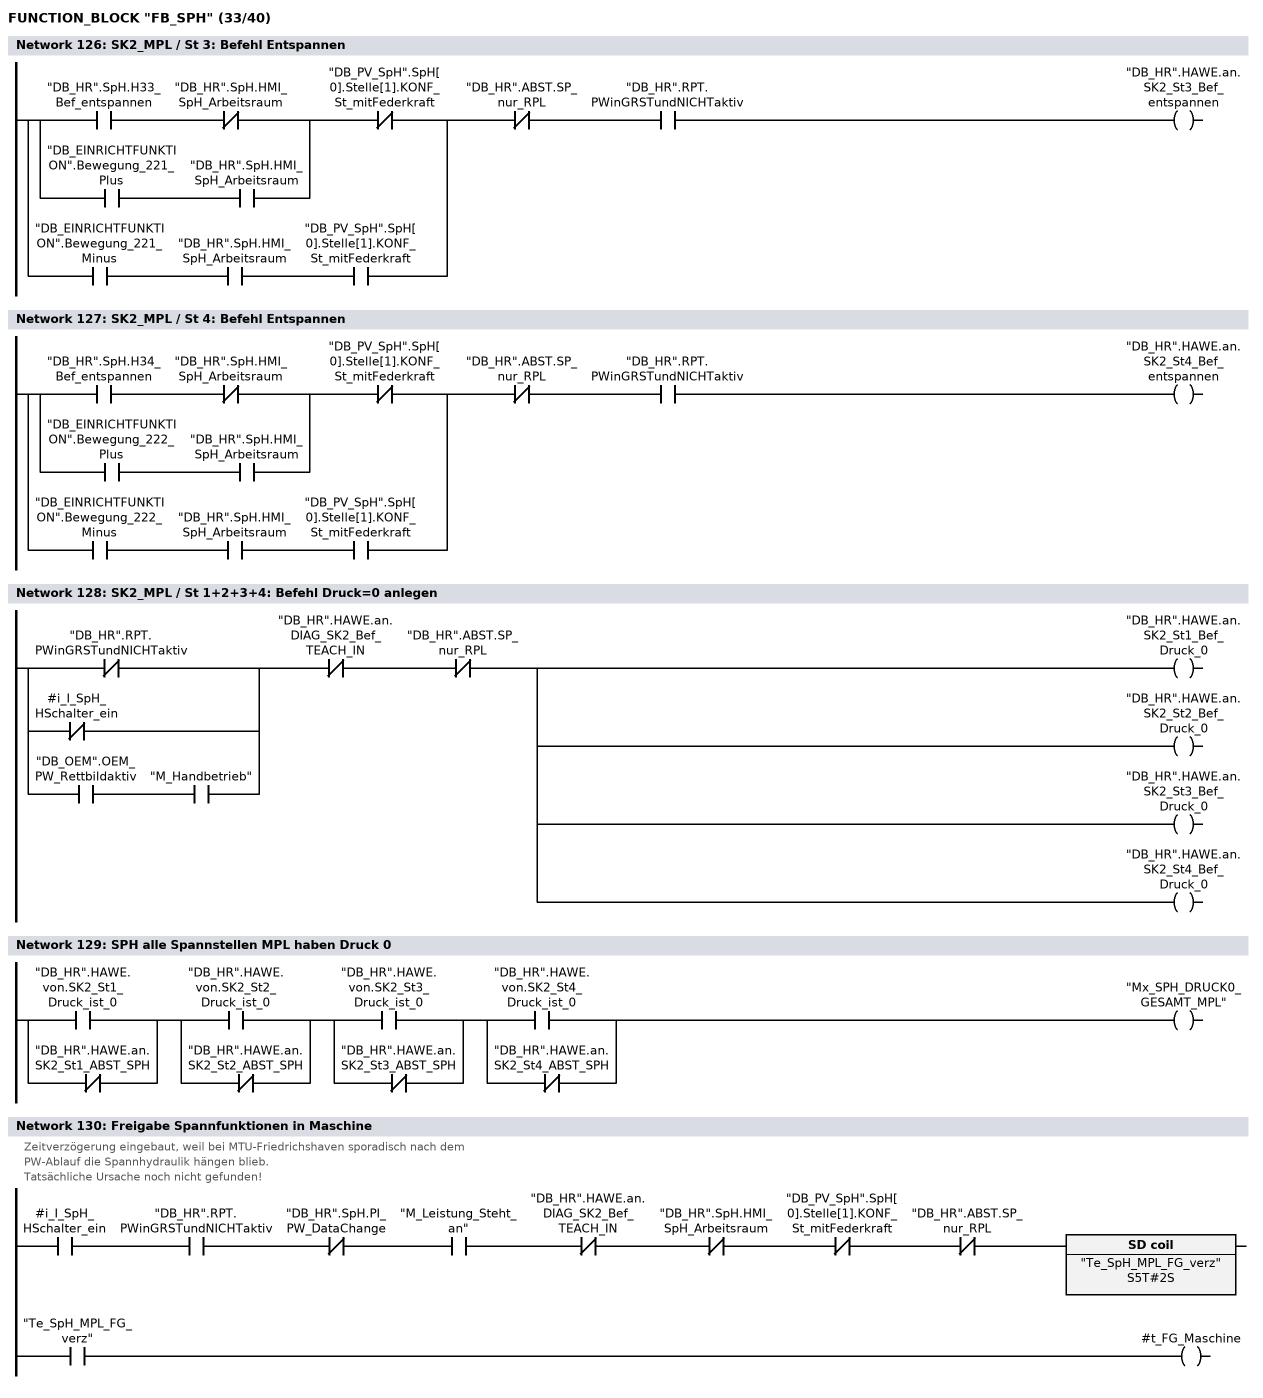

      U(    ;
      U(    ;
      U     "DB_HR".SpH.H33_Bef_entspannen;
      UN    "DB_HR".SpH.HMI_SpH_Arbeitsraum;
      O     ;
      U     "DB_EINRICHTFUNKTION".Bewegung_221_Plus;
      U     "DB_HR".SpH.HMI_SpH_Arbeitsraum;
      )     ;
      UN    "DB_PV_SpH".SpH[0].Stelle[1].KONF_St_mitFederkraft;

      O     ;
      U     "DB_EINRICHTFUNKTION".Bewegung_221_Minus;
      U     "DB_HR".SpH.HMI_SpH_Arbeitsraum;
      U     "DB_PV_SpH".SpH[0].Stelle[1].KONF_St_mitFederkraft;
      )     ;
      UN    "DB_HR".ABST.SP_nur_RPL;
      U     "DB_HR".RPT.PWinGRSTundNICHTaktiv;
      =     "DB_HR".HAWE.an.SK2_St3_Bef_entspannen;
NETWORK
TITLE =SK2_MPL / St 4: Befehl Entspannen

      U(    ;
      U(    ;
      U     "DB_HR".SpH.H34_Bef_entspannen;
      UN    "DB_HR".SpH.HMI_SpH_Arbeitsraum;
      O     ;
      U     "DB_EINRICHTFUNKTION".Bewegung_222_Plus;
      U     "DB_HR".SpH.HMI_SpH_Arbeitsraum;
      )     ;
      UN    "DB_PV_SpH".SpH[0].Stelle[1].KONF_St_mitFederkraft;

      O     ;
      U     "DB_EINRICHTFUNKTION".Bewegung_222_Minus;
      U     "DB_HR".SpH.HMI_SpH_Arbeitsraum;
      U     "DB_PV_SpH".SpH[0].Stelle[1].KONF_St_mitFederkraft;
      )     ;
      UN    "DB_HR".ABST.SP_nur_RPL;
      U     "DB_HR".RPT.PWinGRSTundNICHTaktiv;
      =     "DB_HR".HAWE.an.SK2_St4_Bef_entspannen;
NETWORK
TITLE =SK2_MPL / St 1+2+3+4: Befehl Druck=0 anlegen

      U(    ;
      ON    "DB_HR".RPT.PWinGRSTundNICHTaktiv;
      ON    #i_I_SpH_HSchalter_ein;
      O     ;
      U     "DB_OEM".OEM_PW_Rettbildaktiv;
      U     "M_Handbetrieb";
      )     ;
      UN    "DB_HR".HAWE.an.DIAG_SK2_Bef_TEACH_IN;
      UN    "DB_HR".ABST.SP_nur_RPL;
      =     "DB_HR".HAWE.an.SK2_St1_Bef_Druck_0;
      =     "DB_HR".HAWE.an.SK2_St2_Bef_Druck_0;
      =     "DB_HR".HAWE.an.SK2_St3_Bef_Druck_0;
      =     "DB_HR".HAWE.an.SK2_St4_Bef_Druck_0;
NETWORK
TITLE =SPH alle Spannstellen MPL haben Druck 0

      U(    ;
      O     "DB_HR".HAWE.von.SK2_St1_Druck_ist_0;
      ON    "DB_HR".HAWE.an.SK2_St1_ABST_SPH;
      )     ;
      U(    ;
      O     "DB_HR".HAWE.von.SK2_St2_Druck_ist_0;
      ON    "DB_HR".HAWE.an.SK2_St2_ABST_SPH;
      )     ;
      U(    ;
      O     "DB_HR".HAWE.von.SK2_St3_Druck_ist_0;
      ON    "DB_HR".HAWE.an.SK2_St3_ABST_SPH;
      )     ;
      U(    ;
      O     "DB_HR".HAWE.von.SK2_St4_Druck_ist_0;
      ON    "DB_HR".HAWE.an.SK2_St4_ABST_SPH;
      )     ;
      =     "Mx_SPH_DRUCK0_GESAMT_MPL";
NETWORK
TITLE =Freigabe Spannfunktionen in Maschine
//Zeitverzögerung eingebaut, weil bei MTU-Friedrichshaven sporadisch nach dem
//PW-Ablauf die Spannhydraulik hängen blieb.
//Tatsächliche Ursache noch nicht gefunden!
      U     #i_I_SpH_HSchalter_ein;
      U     "DB_HR".RPT.PWinGRSTundNICHTaktiv;
      UN    "DB_HR".SpH.PI_PW_DataChange;
      U     "M_Leistung_Steht_an";
      UN    "DB_HR".HAWE.an.DIAG_SK2_Bef_TEACH_IN;
      UN    "DB_HR".SpH.HMI_SpH_Arbeitsraum;
      UN    "DB_PV_SpH".SpH[0].Stelle[1].KONF_St_mitFederkraft;
      UN    "DB_HR".ABST.SP_nur_RPL;
      L     S5T#2S;
      SE    "Te_SpH_MPL_FG_verz";
      NOP   0;
      NOP   0;
      NOP   0;
      U     "Te_SpH_MPL_FG_verz";
      =     #t_FG_Maschine;
NETWORK
TITLE =NI Bild SpannHydraulik-Arbeitsraum aktiv
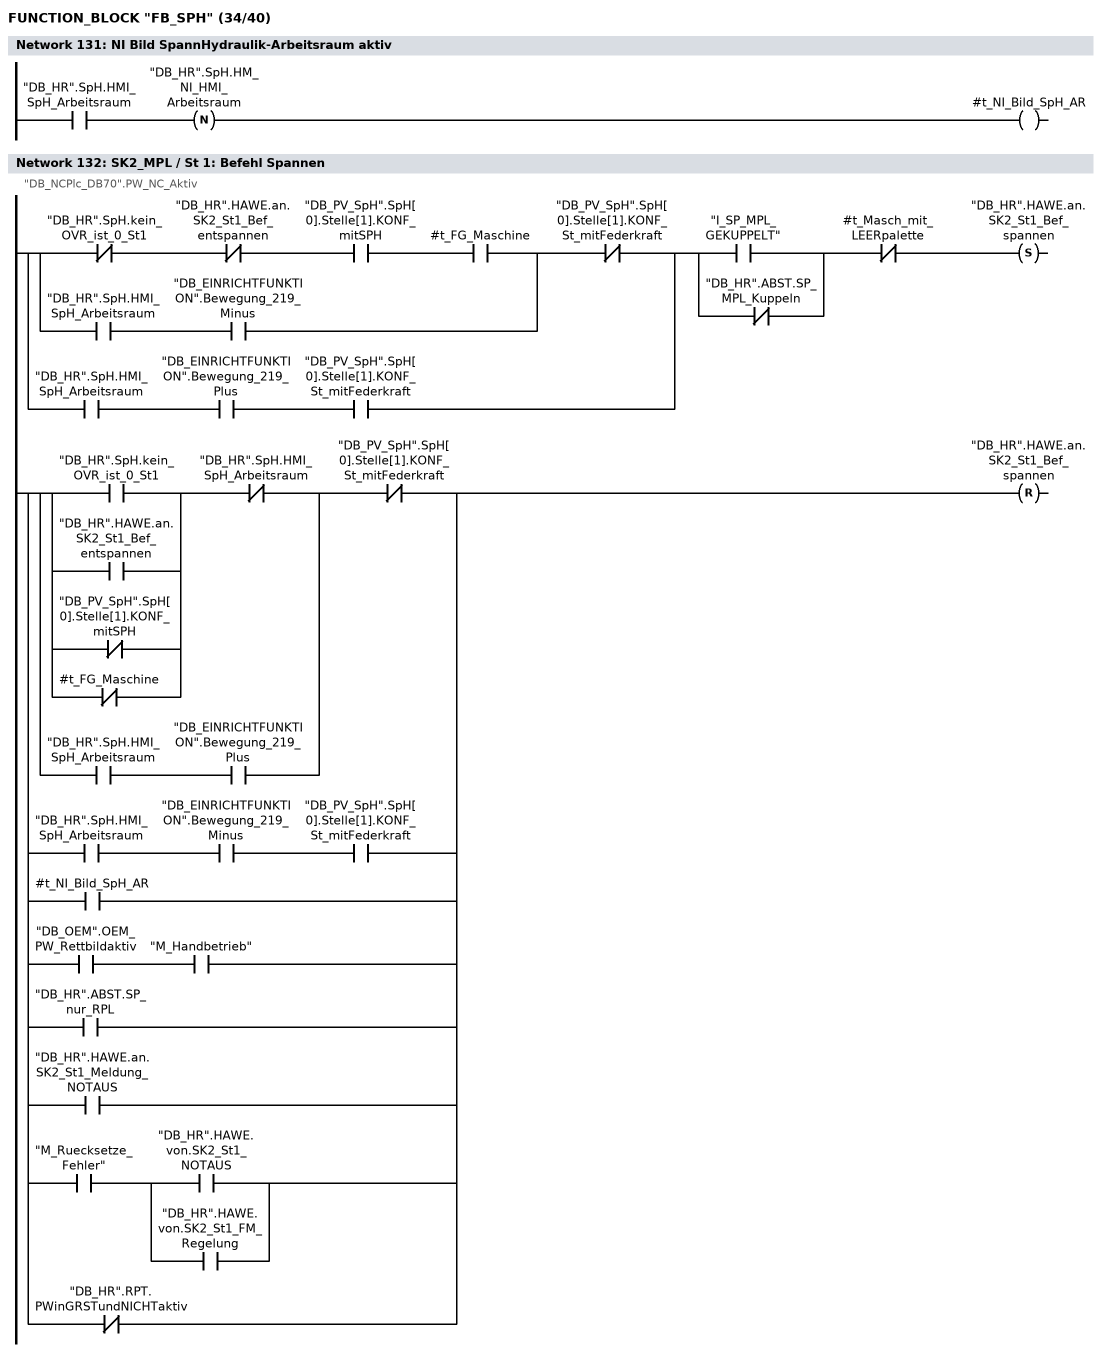

      U     "DB_HR".SpH.HMI_SpH_Arbeitsraum;
      FN    "DB_HR".SpH.HM_NI_HMI_Arbeitsraum;
      =     #t_NI_Bild_SpH_AR;
NETWORK
TITLE =SK2_MPL / St 1: Befehl Spannen
//"DB_NCPlc_DB70".PW_NC_Aktiv
      U(    ;
      U(    ;
      UN    "DB_HR".SpH.kein_OVR_ist_0_St1;
      UN    "DB_HR".HAWE.an.SK2_St1_Bef_entspannen;
      U     "DB_PV_SpH".SpH[0].Stelle[1].KONF_mitSPH;
      U     #t_FG_Maschine;
      O     ;
      U     "DB_HR".SpH.HMI_SpH_Arbeitsraum;
      U     "DB_EINRICHTFUNKTION".Bewegung_219_Minus;
      )     ;
      UN    "DB_PV_SpH".SpH[0].Stelle[1].KONF_St_mitFederkraft;

      O     ;
      U     "DB_HR".SpH.HMI_SpH_Arbeitsraum;
      U     "DB_EINRICHTFUNKTION".Bewegung_219_Plus;
      U     "DB_PV_SpH".SpH[0].Stelle[1].KONF_St_mitFederkraft;
      )     ;
      U(    ;
      O     "I_SP_MPL_GEKUPPELT";
      ON    "DB_HR".ABST.SP_MPL_Kuppeln;
      )     ;
      UN    #t_Masch_mit_LEERpalette;

      S     "DB_HR".HAWE.an.SK2_St1_Bef_spannen;
      U(    ;
      U(    ;
      U(    ;
      O     "DB_HR".SpH.kein_OVR_ist_0_St1;
      O     "DB_HR".HAWE.an.SK2_St1_Bef_entspannen;
      ON    "DB_PV_SpH".SpH[0].Stelle[1].KONF_mitSPH;
      ON    #t_FG_Maschine;
      )     ;

      UN    "DB_HR".SpH.HMI_SpH_Arbeitsraum;
      O     ;
      U     "DB_HR".SpH.HMI_SpH_Arbeitsraum;
      U     "DB_EINRICHTFUNKTION".Bewegung_219_Plus;
      )     ;

      UN    "DB_PV_SpH".SpH[0].Stelle[1].KONF_St_mitFederkraft;
      O     ;
      U     "DB_HR".SpH.HMI_SpH_Arbeitsraum;
      U     "DB_EINRICHTFUNKTION".Bewegung_219_Minus;

      U     "DB_PV_SpH".SpH[0].Stelle[1].KONF_St_mitFederkraft;
      O     #t_NI_Bild_SpH_AR;
      O     ;
      U     "DB_OEM".OEM_PW_Rettbildaktiv;
      U     "M_Handbetrieb";
      O     "DB_HR".ABST.SP_nur_RPL;
      O     "DB_HR".HAWE.an.SK2_St1_Meldung_NOTAUS;
      O     ;
      U     "M_Ruecksetze_Fehler";
      U(    ;
      O     "DB_HR".HAWE.von.SK2_St1_NOTAUS;
      O     "DB_HR".HAWE.von.SK2_St1_FM_Regelung;
      )     ;
      ON    "DB_HR".RPT.PWinGRSTundNICHTaktiv;
      )     ;
      R     "DB_HR".HAWE.an.SK2_St1_Bef_spannen;
      NOP   0;
NETWORK
TITLE =SK2_MPL / St 2: Befehl Spannen
//"DB_NCPlc_DB70".PW_NC_Aktiv
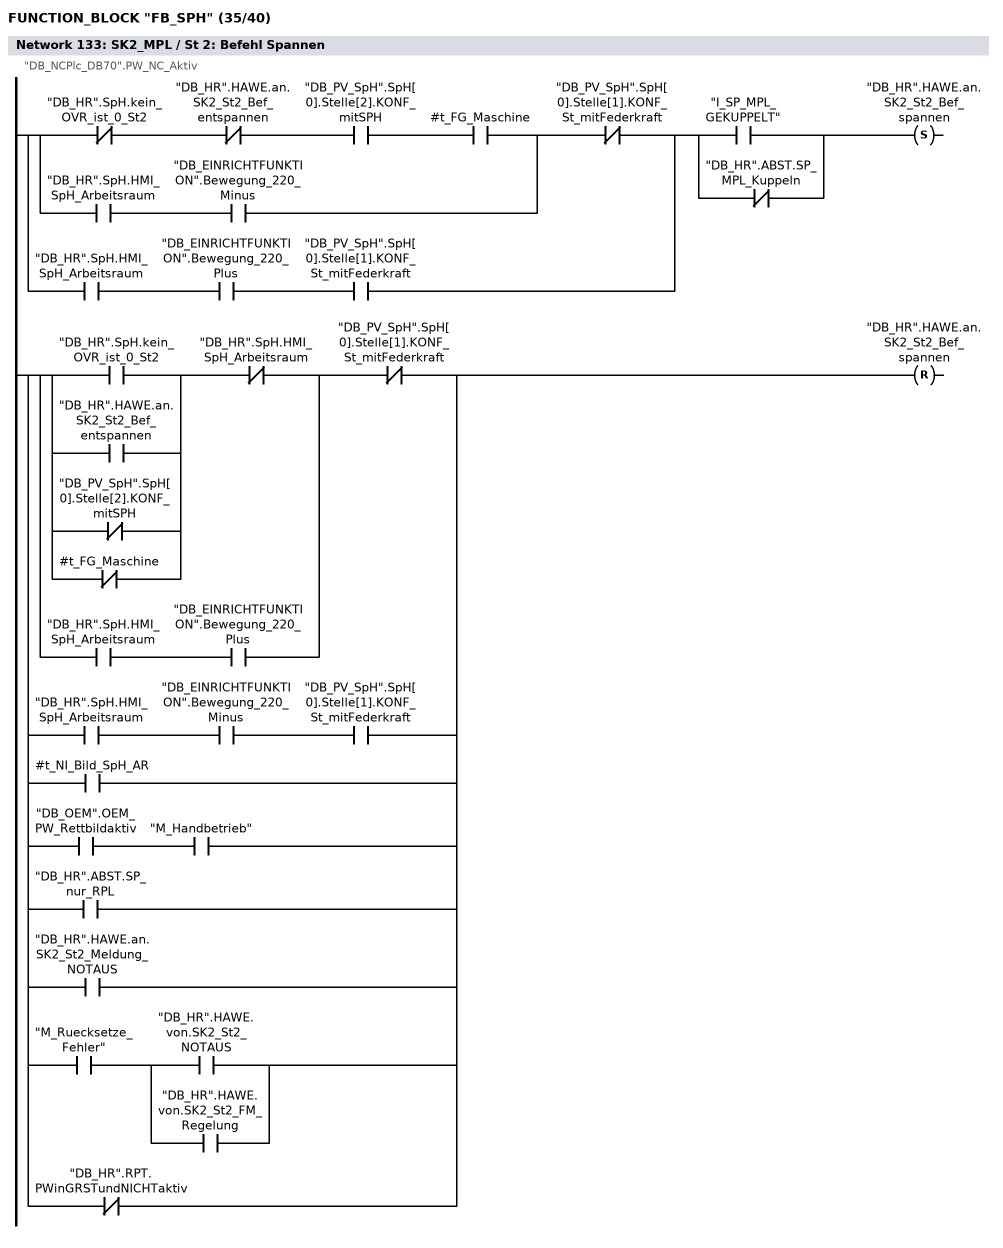
      U(    ;
      U(    ;
      UN    "DB_HR".SpH.kein_OVR_ist_0_St2;
      UN    "DB_HR".HAWE.an.SK2_St2_Bef_entspannen;
      U     "DB_PV_SpH".SpH[0].Stelle[2].KONF_mitSPH;
      U     #t_FG_Maschine;
      O     ;
      U     "DB_HR".SpH.HMI_SpH_Arbeitsraum;
      U     "DB_EINRICHTFUNKTION".Bewegung_220_Minus;
      )     ;
      UN    "DB_PV_SpH".SpH[0].Stelle[1].KONF_St_mitFederkraft;

      O     ;
      U     "DB_HR".SpH.HMI_SpH_Arbeitsraum;
      U     "DB_EINRICHTFUNKTION".Bewegung_220_Plus;
      U     "DB_PV_SpH".SpH[0].Stelle[1].KONF_St_mitFederkraft;
      )     ;
      U(    ;
      O     "I_SP_MPL_GEKUPPELT";
      ON    "DB_HR".ABST.SP_MPL_Kuppeln;
      )     ;
      S     "DB_HR".HAWE.an.SK2_St2_Bef_spannen;

      U(    ;
      U(    ;
      U(    ;
      O     "DB_HR".SpH.kein_OVR_ist_0_St2;
      O     "DB_HR".HAWE.an.SK2_St2_Bef_entspannen;
      ON    "DB_PV_SpH".SpH[0].Stelle[2].KONF_mitSPH;
      ON    #t_FG_Maschine;
      )     ;
      UN    "DB_HR".SpH.HMI_SpH_Arbeitsraum;
      O     ;
      U     "DB_HR".SpH.HMI_SpH_Arbeitsraum;
      U     "DB_EINRICHTFUNKTION".Bewegung_220_Plus;
      )     ;
      UN    "DB_PV_SpH".SpH[0].Stelle[1].KONF_St_mitFederkraft;
      O     ;
      U     "DB_HR".SpH.HMI_SpH_Arbeitsraum;
      U     "DB_EINRICHTFUNKTION".Bewegung_220_Minus;
      U     "DB_PV_SpH".SpH[0].Stelle[1].KONF_St_mitFederkraft;
      O     #t_NI_Bild_SpH_AR;
      O     ;
      U     "DB_OEM".OEM_PW_Rettbildaktiv;
      U     "M_Handbetrieb";
      O     "DB_HR".ABST.SP_nur_RPL;
      O     "DB_HR".HAWE.an.SK2_St2_Meldung_NOTAUS;
      O     ;
      U     "M_Ruecksetze_Fehler";
      U(    ;
      O     "DB_HR".HAWE.von.SK2_St2_NOTAUS;
      O     "DB_HR".HAWE.von.SK2_St2_FM_Regelung;
      )     ;
      ON    "DB_HR".RPT.PWinGRSTundNICHTaktiv;
      )     ;
      R     "DB_HR".HAWE.an.SK2_St2_Bef_spannen;
      NOP   0;
NETWORK
TITLE =SK2_MPL / St 3: Befehl Spannen
//"DB_NCPlc_DB70".PW_NC_Aktiv
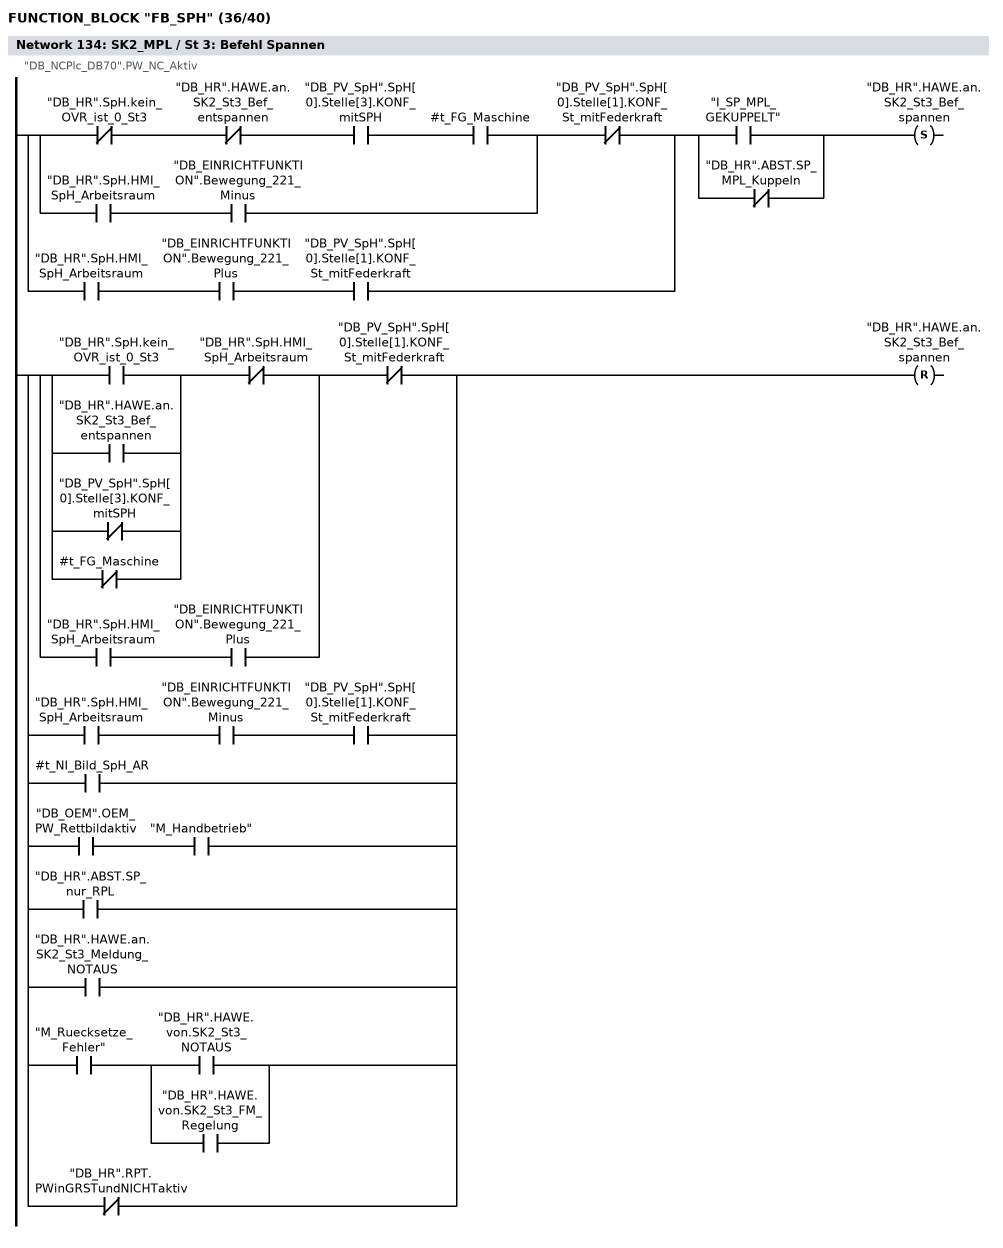
      U(    ;
      U(    ;
      UN    "DB_HR".SpH.kein_OVR_ist_0_St3;
      UN    "DB_HR".HAWE.an.SK2_St3_Bef_entspannen;
      U     "DB_PV_SpH".SpH[0].Stelle[3].KONF_mitSPH;
      U     #t_FG_Maschine;
      O     ;
      U     "DB_HR".SpH.HMI_SpH_Arbeitsraum;
      U     "DB_EINRICHTFUNKTION".Bewegung_221_Minus;
      )     ;
      UN    "DB_PV_SpH".SpH[0].Stelle[1].KONF_St_mitFederkraft;
      O     ;
      U     "DB_HR".SpH.HMI_SpH_Arbeitsraum;
      U     "DB_EINRICHTFUNKTION".Bewegung_221_Plus;
      U     "DB_PV_SpH".SpH[0].Stelle[1].KONF_St_mitFederkraft;
      )     ;
      U(    ;
      O     "I_SP_MPL_GEKUPPELT";
      ON    "DB_HR".ABST.SP_MPL_Kuppeln;
      )     ;
      S     "DB_HR".HAWE.an.SK2_St3_Bef_spannen;
      U(    ;
      U(    ;
      U(    ;
      O     "DB_HR".SpH.kein_OVR_ist_0_St3;
      O     "DB_HR".HAWE.an.SK2_St3_Bef_entspannen;
      ON    "DB_PV_SpH".SpH[0].Stelle[3].KONF_mitSPH;
      ON    #t_FG_Maschine;
      )     ;
      UN    "DB_HR".SpH.HMI_SpH_Arbeitsraum;
      O     ;
      U     "DB_HR".SpH.HMI_SpH_Arbeitsraum;
      U     "DB_EINRICHTFUNKTION".Bewegung_221_Plus;
      )     ;
      UN    "DB_PV_SpH".SpH[0].Stelle[1].KONF_St_mitFederkraft;
      O     ;
      U     "DB_HR".SpH.HMI_SpH_Arbeitsraum;
      U     "DB_EINRICHTFUNKTION".Bewegung_221_Minus;
      U     "DB_PV_SpH".SpH[0].Stelle[1].KONF_St_mitFederkraft;
      O     #t_NI_Bild_SpH_AR;
      O     ;
      U     "DB_OEM".OEM_PW_Rettbildaktiv;
      U     "M_Handbetrieb";
      O     "DB_HR".ABST.SP_nur_RPL;
      O     "DB_HR".HAWE.an.SK2_St3_Meldung_NOTAUS;
      O     ;
      U     "M_Ruecksetze_Fehler";
      U(    ;
      O     "DB_HR".HAWE.von.SK2_St3_NOTAUS;
      O     "DB_HR".HAWE.von.SK2_St3_FM_Regelung;
      )     ;
      ON    "DB_HR".RPT.PWinGRSTundNICHTaktiv;
      )     ;
      R     "DB_HR".HAWE.an.SK2_St3_Bef_spannen;
      NOP   0;
NETWORK
TITLE =SK2_MPL / St 4: Befehl Spannen
//"DB_NCPlc_DB70".PW_NC_Aktiv
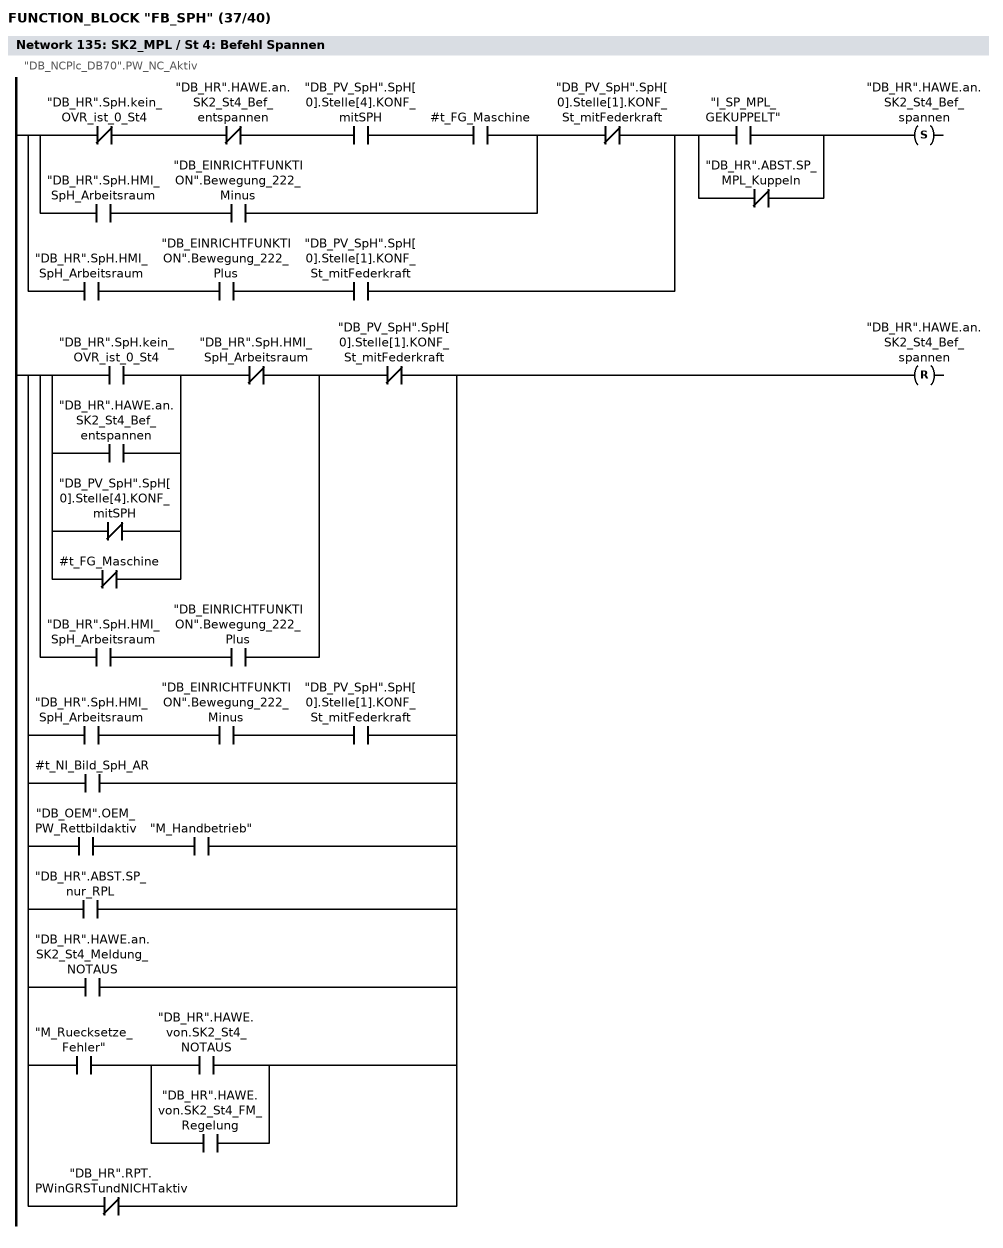
      U(    ;
      U(    ;
      UN    "DB_HR".SpH.kein_OVR_ist_0_St4;
      UN    "DB_HR".HAWE.an.SK2_St4_Bef_entspannen;
      U     "DB_PV_SpH".SpH[0].Stelle[4].KONF_mitSPH;
      U     #t_FG_Maschine;
      O     ;
      U     "DB_HR".SpH.HMI_SpH_Arbeitsraum;
      U     "DB_EINRICHTFUNKTION".Bewegung_222_Minus;
      )     ;
      UN    "DB_PV_SpH".SpH[0].Stelle[1].KONF_St_mitFederkraft;
      O     ;
      U     "DB_HR".SpH.HMI_SpH_Arbeitsraum;
      U     "DB_EINRICHTFUNKTION".Bewegung_222_Plus;
      U     "DB_PV_SpH".SpH[0].Stelle[1].KONF_St_mitFederkraft;
      )     ;
      U(    ;
      O     "I_SP_MPL_GEKUPPELT";
      ON    "DB_HR".ABST.SP_MPL_Kuppeln;
      )     ;
      S     "DB_HR".HAWE.an.SK2_St4_Bef_spannen;
      U(    ;
      U(    ;
      U(    ;
      O     "DB_HR".SpH.kein_OVR_ist_0_St4;
      O     "DB_HR".HAWE.an.SK2_St4_Bef_entspannen;
      ON    "DB_PV_SpH".SpH[0].Stelle[4].KONF_mitSPH;
      ON    #t_FG_Maschine;
      )     ;
      UN    "DB_HR".SpH.HMI_SpH_Arbeitsraum;
      O     ;
      U     "DB_HR".SpH.HMI_SpH_Arbeitsraum;
      U     "DB_EINRICHTFUNKTION".Bewegung_222_Plus;
      )     ;
      UN    "DB_PV_SpH".SpH[0].Stelle[1].KONF_St_mitFederkraft;
      O     ;
      U     "DB_HR".SpH.HMI_SpH_Arbeitsraum;
      U     "DB_EINRICHTFUNKTION".Bewegung_222_Minus;
      U     "DB_PV_SpH".SpH[0].Stelle[1].KONF_St_mitFederkraft;
      O     #t_NI_Bild_SpH_AR;
      O     ;
      U     "DB_OEM".OEM_PW_Rettbildaktiv;
      U     "M_Handbetrieb";
      O     "DB_HR".ABST.SP_nur_RPL;
      O     "DB_HR".HAWE.an.SK2_St4_Meldung_NOTAUS;
      O     ;
      U     "M_Ruecksetze_Fehler";
      U(    ;
      O     "DB_HR".HAWE.von.SK2_St4_NOTAUS;
      O     "DB_HR".HAWE.von.SK2_St4_FM_Regelung;
      )     ;
      ON    "DB_HR".RPT.PWinGRSTundNICHTaktiv;
      )     ;
      R     "DB_HR".HAWE.an.SK2_St4_Bef_spannen;
      NOP   0;
NETWORK
TITLE =SK2_MPL / St 1+2+3+4: Meldung NOTAUS
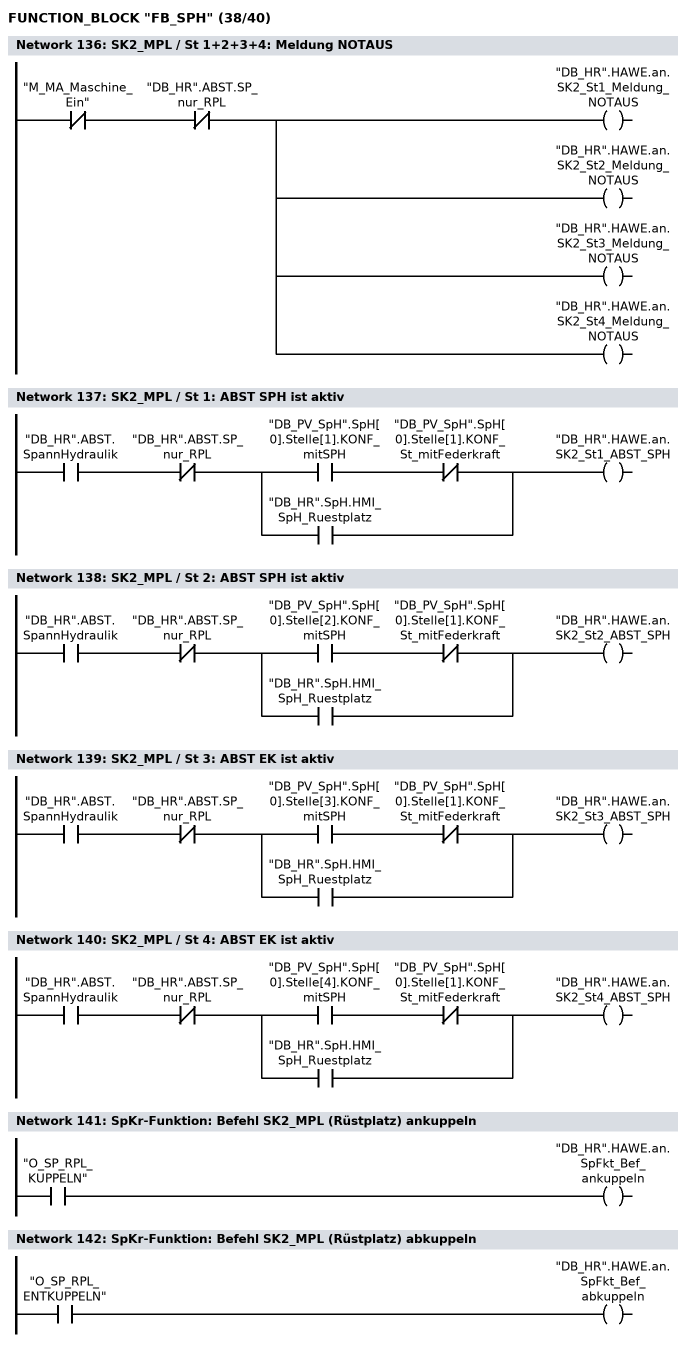

      UN    "M_MA_Maschine_Ein";
      UN    "DB_HR".ABST.SP_nur_RPL;
      =     "DB_HR".HAWE.an.SK2_St1_Meldung_NOTAUS;
      =     "DB_HR".HAWE.an.SK2_St2_Meldung_NOTAUS;
      =     "DB_HR".HAWE.an.SK2_St3_Meldung_NOTAUS;
      =     "DB_HR".HAWE.an.SK2_St4_Meldung_NOTAUS;
NETWORK
TITLE =SK2_MPL / St 1: ABST SPH ist aktiv

      U     "DB_HR".ABST.SpannHydraulik;
      UN    "DB_HR".ABST.SP_nur_RPL;
      U(    ;
      U     "DB_PV_SpH".SpH[0].Stelle[1].KONF_mitSPH;
      UN    "DB_PV_SpH".SpH[0].Stelle[1].KONF_St_mitFederkraft;
      O     "DB_HR".SpH.HMI_SpH_Ruestplatz;
      )     ;
      =     "DB_HR".HAWE.an.SK2_St1_ABST_SPH;
NETWORK
TITLE =SK2_MPL / St 2: ABST SPH ist aktiv

      U     "DB_HR".ABST.SpannHydraulik;
      UN    "DB_HR".ABST.SP_nur_RPL;
      U(    ;
      U     "DB_PV_SpH".SpH[0].Stelle[2].KONF_mitSPH;
      UN    "DB_PV_SpH".SpH[0].Stelle[1].KONF_St_mitFederkraft;
      O     "DB_HR".SpH.HMI_SpH_Ruestplatz;
      )     ;
      =     "DB_HR".HAWE.an.SK2_St2_ABST_SPH;
NETWORK
TITLE =SK2_MPL / St 3: ABST EK ist aktiv

      U     "DB_HR".ABST.SpannHydraulik;
      UN    "DB_HR".ABST.SP_nur_RPL;
      U(    ;
      U     "DB_PV_SpH".SpH[0].Stelle[3].KONF_mitSPH;
      UN    "DB_PV_SpH".SpH[0].Stelle[1].KONF_St_mitFederkraft;
      O     "DB_HR".SpH.HMI_SpH_Ruestplatz;
      )     ;
      =     "DB_HR".HAWE.an.SK2_St3_ABST_SPH;
NETWORK
TITLE =SK2_MPL / St 4: ABST EK ist aktiv

      U     "DB_HR".ABST.SpannHydraulik;
      UN    "DB_HR".ABST.SP_nur_RPL;
      U(    ;
      U     "DB_PV_SpH".SpH[0].Stelle[4].KONF_mitSPH;
      UN    "DB_PV_SpH".SpH[0].Stelle[1].KONF_St_mitFederkraft;
      O     "DB_HR".SpH.HMI_SpH_Ruestplatz;
      )     ;
      =     "DB_HR".HAWE.an.SK2_St4_ABST_SPH;
NETWORK
TITLE =SpKr-Funktion: Befehl SK2_MPL (Rüstplatz) ankuppeln

      U     "O_SP_RPL_KUPPELN";
      =     "DB_HR".HAWE.an.SpFkt_Bef_ankuppeln;
NETWORK
TITLE =SpKr-Funktion: Befehl SK2_MPL (Rüstplatz) abkuppeln

      U     "O_SP_RPL_ENTKUPPELN";
      =     "DB_HR".HAWE.an.SpFkt_Bef_abkuppeln;
NETWORK
TITLE =HMI-Anzeige: Rüstplatz Teachen
//Bild-Nr: 41 Zeile: 2
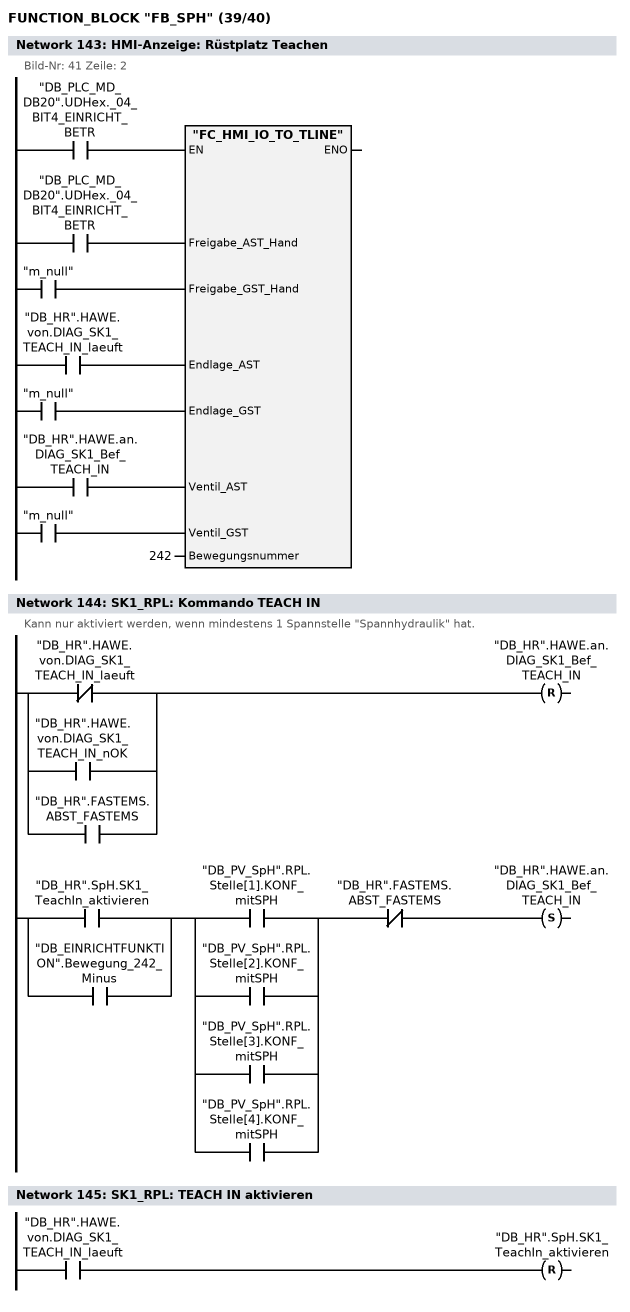
      U     "DB_PLC_MD_DB20".UDHex._04_BIT4_EINRICHT_BETR;
      =     L     18.0;
      BLD   103;
      U     "m_null";
      =     L     18.1;
      BLD   103;
      U     "DB_HR".HAWE.von.DIAG_SK1_TEACH_IN_laeuft;
      =     L     18.2;
      BLD   103;
      U     "m_null";
      =     L     18.3;
      BLD   103;
      U     "DB_HR".HAWE.an.DIAG_SK1_Bef_TEACH_IN;
      =     L     18.4;
      BLD   103;
      U     "m_null";
      =     L     18.5;
      BLD   103;
      U     "DB_PLC_MD_DB20".UDHex._04_BIT4_EINRICHT_BETR;
      SPBNB _012;
      CALL "FC_HMI_IO_TO_TLINE" (
           Freigabe_AST_Hand        := L     18.0,
           Freigabe_GST_Hand        := L     18.1,
           Endlage_AST              := L     18.2,
           Endlage_GST              := L     18.3,
           Ventil_AST               := L     18.4,
           Ventil_GST               := L     18.5,
           Bewegungsnummer          := 242);
_012: NOP   0;
NETWORK
TITLE =SK1_RPL: Kommando TEACH IN
//Kann nur aktiviert werden, wenn mindestens 1 Spannstelle "Spannhydraulik" hat.
      U(    ;
      ON    "DB_HR".HAWE.von.DIAG_SK1_TEACH_IN_laeuft;
      O     "DB_HR".HAWE.von.DIAG_SK1_TEACH_IN_nOK;
      O     "DB_HR".FASTEMS.ABST_FASTEMS;
      )     ;
      R     "DB_HR".HAWE.an.DIAG_SK1_Bef_TEACH_IN;
      U(    ;
      O     "DB_HR".SpH.SK1_TeachIn_aktivieren;
      O     "DB_EINRICHTFUNKTION".Bewegung_242_Minus;
      )     ;
      U(    ;
      O     "DB_PV_SpH".RPL.Stelle[1].KONF_mitSPH;
      O     "DB_PV_SpH".RPL.Stelle[2].KONF_mitSPH;
      O     "DB_PV_SpH".RPL.Stelle[3].KONF_mitSPH;
      O     "DB_PV_SpH".RPL.Stelle[4].KONF_mitSPH;
      )     ;
      UN    "DB_HR".FASTEMS.ABST_FASTEMS;
      S     "DB_HR".HAWE.an.DIAG_SK1_Bef_TEACH_IN;
      NOP   0;
NETWORK
TITLE =SK1_RPL: TEACH IN aktivieren

      U     "DB_HR".HAWE.von.DIAG_SK1_TEACH_IN_laeuft;
      R     "DB_HR".SpH.SK1_TeachIn_aktivieren;
NETWORK
TITLE =HMI-Anzeige: Maschinenraum Teachen
//Bild-Nr: 41 Zeile: 3
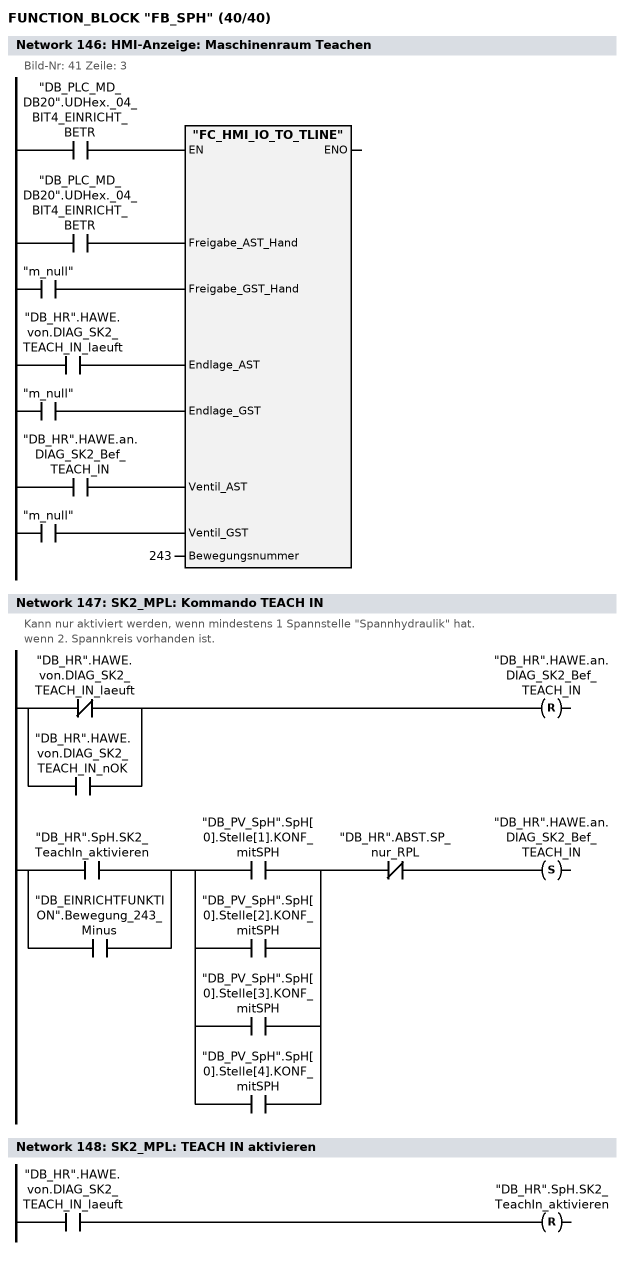
      U     "DB_PLC_MD_DB20".UDHex._04_BIT4_EINRICHT_BETR;
      =     L     18.0;
      BLD   103;
      U     "m_null";
      =     L     18.1;
      BLD   103;
      U     "DB_HR".HAWE.von.DIAG_SK2_TEACH_IN_laeuft;
      =     L     18.2;
      BLD   103;
      U     "m_null";
      =     L     18.3;
      BLD   103;
      U     "DB_HR".HAWE.an.DIAG_SK2_Bef_TEACH_IN;
      =     L     18.4;
      BLD   103;
      U     "m_null";
      =     L     18.5;
      BLD   103;
      U     "DB_PLC_MD_DB20".UDHex._04_BIT4_EINRICHT_BETR;
      SPBNB _013;
      CALL "FC_HMI_IO_TO_TLINE" (
           Freigabe_AST_Hand        := L     18.0,
           Freigabe_GST_Hand        := L     18.1,
           Endlage_AST              := L     18.2,
           Endlage_GST              := L     18.3,
           Ventil_AST               := L     18.4,
           Ventil_GST               := L     18.5,
           Bewegungsnummer          := 243);
_013: NOP   0;
NETWORK
TITLE =SK2_MPL: Kommando TEACH IN
//Kann nur aktiviert werden, wenn mindestens 1 Spannstelle "Spannhydraulik" hat.
//                           wenn 2. Spannkreis vorhanden ist.
      U(    ;
      ON    "DB_HR".HAWE.von.DIAG_SK2_TEACH_IN_laeuft;
      O     "DB_HR".HAWE.von.DIAG_SK2_TEACH_IN_nOK;
      )     ;
      R     "DB_HR".HAWE.an.DIAG_SK2_Bef_TEACH_IN;
      U(    ;
      O     "DB_HR".SpH.SK2_TeachIn_aktivieren;
      O     "DB_EINRICHTFUNKTION".Bewegung_243_Minus;
      )     ;
      U(    ;
      O     "DB_PV_SpH".SpH[0].Stelle[1].KONF_mitSPH;
      O     "DB_PV_SpH".SpH[0].Stelle[2].KONF_mitSPH;
      O     "DB_PV_SpH".SpH[0].Stelle[3].KONF_mitSPH;
      O     "DB_PV_SpH".SpH[0].Stelle[4].KONF_mitSPH;
      )     ;
      UN    "DB_HR".ABST.SP_nur_RPL;
      S     "DB_HR".HAWE.an.DIAG_SK2_Bef_TEACH_IN;
      NOP   0;
NETWORK
TITLE =SK2_MPL: TEACH IN aktivieren

      U     "DB_HR".HAWE.von.DIAG_SK2_TEACH_IN_laeuft;
      R     "DB_HR".SpH.SK2_TeachIn_aktivieren;
NETWORK
TITLE =Diagnose: Lebenszeichen-Überwachung

      U     "m_takt_0,5sec.";
      FP    "DB_HR".SpH.HM_PI_Takt;
      SPBN  LBZ;
      UN    "DB_HR".HAWE.an.DIAG_Lebenszeichen;
      =     "DB_HR".HAWE.an.DIAG_Lebenszeichen;
LBZ:  NOP   0;
NETWORK
TITLE =702349 "WAR, Lebenszeichen ProfiBus-HAWE-Box fehlt!"

      U(    ;
      U     "DB_HR".ABST.SpannHydraulik;
      UN    "DB_CONFIG".ABST.SPH_VORBEREITET;
      UN    "DB_HR".HAWE.von.DIAG_Lebenszeichen;
      U     "M_MA_Maschine_Ein";
      L     S5T#2S;
      SE    "Te_HAWE_Lebenszeichen";
      NOP   0;
      NOP   0;
      NOP   0;
      U     "Te_HAWE_Lebenszeichen";
      )     ;
      =     #t_LZ_HAWE_niO;
      U     #t_LZ_HAWE_niO;
      S     "DB_FEHLERMELDUNG".WARNUNG4._702349;
      UN    #t_LZ_HAWE_niO;
      U     "M_Ruecksetze_Fehler";
      R     "DB_FEHLERMELDUNG".WARNUNG4._702349;
      NOP   0;
NETWORK
TITLE =INT_165: Tol-Fenster(+/-) "Druck erreicht" (initial: 3bar)
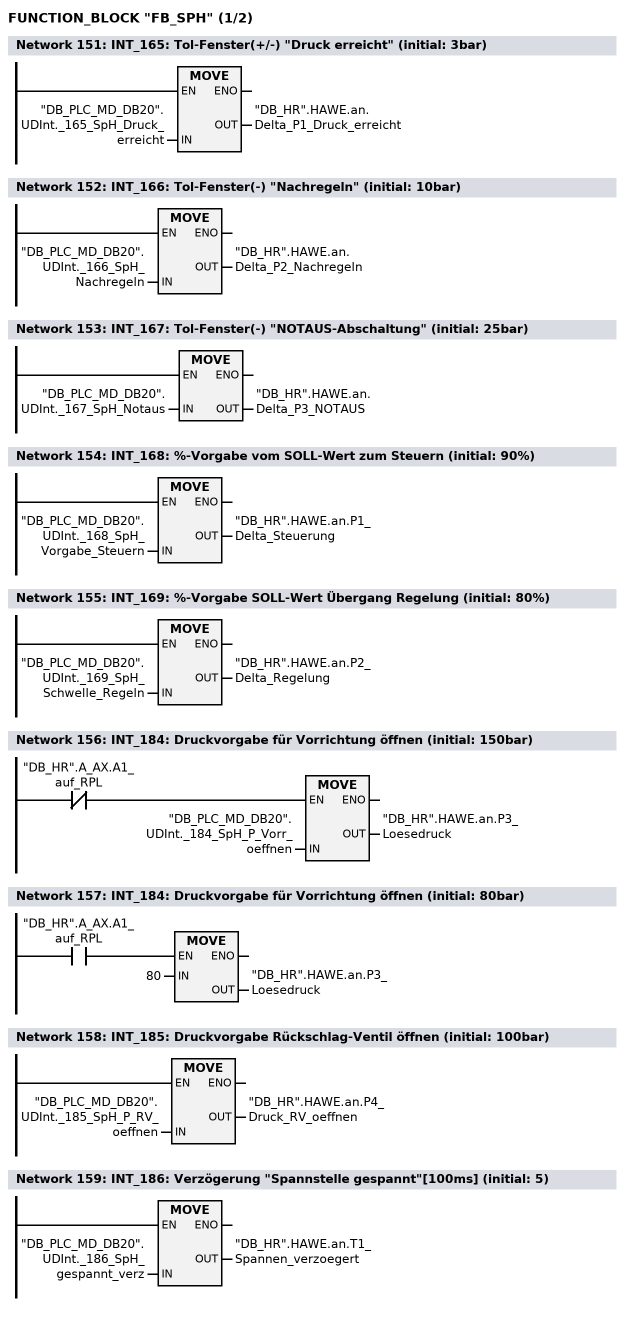

      L     "DB_PLC_MD_DB20".UDInt._165_SpH_Druck_erreicht;
      T     "DB_HR".HAWE.an.Delta_P1_Druck_erreicht;
      NOP   0;
NETWORK
TITLE =INT_166: Tol-Fenster(-) "Nachregeln" (initial: 10bar)

      L     "DB_PLC_MD_DB20".UDInt._166_SpH_Nachregeln;
      T     "DB_HR".HAWE.an.Delta_P2_Nachregeln;
      NOP   0;
NETWORK
TITLE =INT_167: Tol-Fenster(-) "NOTAUS-Abschaltung" (initial: 25bar)

      L     "DB_PLC_MD_DB20".UDInt._167_SpH_Notaus;
      T     "DB_HR".HAWE.an.Delta_P3_NOTAUS;
      NOP   0;
NETWORK
TITLE =INT_168: %-Vorgabe vom SOLL-Wert zum Steuern (initial: 90%)

      L     "DB_PLC_MD_DB20".UDInt._168_SpH_Vorgabe_Steuern;
      T     "DB_HR".HAWE.an.P1_Delta_Steuerung;
      NOP   0;
NETWORK
TITLE =INT_169: %-Vorgabe SOLL-Wert Übergang Regelung (initial: 80%)

      L     "DB_PLC_MD_DB20".UDInt._169_SpH_Schwelle_Regeln;
      T     "DB_HR".HAWE.an.P2_Delta_Regelung;
      NOP   0;
NETWORK
TITLE =INT_184: Druckvorgabe für Vorrichtung öffnen (initial: 150bar)

      UN    "DB_HR".A_AX.A1_auf_RPL;
      SPBNB _014;
      L     "DB_PLC_MD_DB20".UDInt._184_SpH_P_Vorr_oeffnen;
      T     "DB_HR".HAWE.an.P3_Loesedruck;
_014: NOP   0;
NETWORK
TITLE =INT_184: Druckvorgabe für Vorrichtung öffnen (initial: 80bar)

      U     "DB_HR".A_AX.A1_auf_RPL;
      SPBNB _015;
      L     80;
      T     "DB_HR".HAWE.an.P3_Loesedruck;
_015: NOP   0;
NETWORK
TITLE =INT_185: Druckvorgabe Rückschlag-Ventil öffnen (initial: 100bar)

      L     "DB_PLC_MD_DB20".UDInt._185_SpH_P_RV_oeffnen;
      T     "DB_HR".HAWE.an.P4_Druck_RV_oeffnen;
      NOP   0;
NETWORK
TITLE =INT_186: Verzögerung "Spannstelle gespannt"[100ms] (initial: 5)

      L     "DB_PLC_MD_DB20".UDInt._186_SpH_gespannt_verz;
      T     "DB_HR".HAWE.an.T1_Spannen_verzoegert;
      NOP   0;
NETWORK
TITLE =INT_187: Laufzeit "Rückschlag-Ventil öffnen"[100ms](initial: 10)
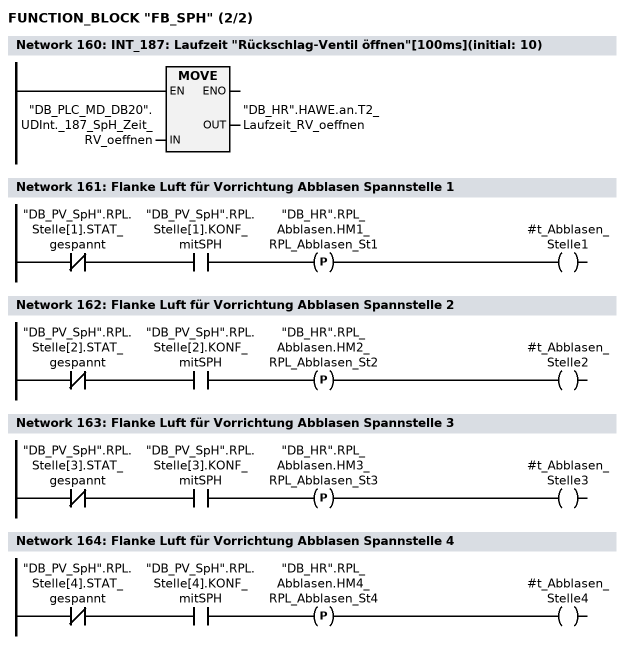

      L     "DB_PLC_MD_DB20".UDInt._187_SpH_Zeit_RV_oeffnen;
      T     "DB_HR".HAWE.an.T2_Laufzeit_RV_oeffnen;
      NOP   0;
NETWORK
TITLE =Flanke Luft für Vorrichtung Abblasen Spannstelle 1

      UN    "DB_PV_SpH".RPL.Stelle[1].STAT_gespannt;
      U     "DB_PV_SpH".RPL.Stelle[1].KONF_mitSPH;
      FP    "DB_HR".RPL_Abblasen.HM1_RPL_Abblasen_St1;
      =     #t_Abblasen_Stelle1;
NETWORK
TITLE =Flanke Luft für Vorrichtung Abblasen Spannstelle 2

      UN    "DB_PV_SpH".RPL.Stelle[2].STAT_gespannt;
      U     "DB_PV_SpH".RPL.Stelle[2].KONF_mitSPH;
      FP    "DB_HR".RPL_Abblasen.HM2_RPL_Abblasen_St2;
      =     #t_Abblasen_Stelle2;
NETWORK
TITLE =Flanke Luft für Vorrichtung Abblasen Spannstelle 3

      UN    "DB_PV_SpH".RPL.Stelle[3].STAT_gespannt;
      U     "DB_PV_SpH".RPL.Stelle[3].KONF_mitSPH;
      FP    "DB_HR".RPL_Abblasen.HM3_RPL_Abblasen_St3;
      =     #t_Abblasen_Stelle3;
NETWORK
TITLE =Flanke Luft für Vorrichtung Abblasen Spannstelle 4

      UN    "DB_PV_SpH".RPL.Stelle[4].STAT_gespannt;
      U     "DB_PV_SpH".RPL.Stelle[4].KONF_mitSPH;
      FP    "DB_HR".RPL_Abblasen.HM4_RPL_Abblasen_St4;
      =     #t_Abblasen_Stelle4;
NETWORK
TITLE =Zeit-Funktion: Spannstelle abblasen in [s]
//DB700.DBB21: "DB_CONFIG".SP.RPL_Spannstelle_abblasen in [s]
      U(    ;
      U(    ;
      U(    ;
      U(    ;
      O     #t_Abblasen_Stelle1;
      O     #t_Abblasen_Stelle2;
      O     #t_Abblasen_Stelle3;
      O     #t_Abblasen_Stelle4;
      )     ;
      SPBNB _016;
      L     "DB_CONFIG".SP.RPL_Spannstelle_abblasen;
      ITB   ;
      T     #t_zeit_Abblasen;
      UN    OV;
      SAVE  ;
      CLR   ;
_016: U     BIE;
      )     ;
      SPBNB _017;
      L     #t_zeit_Abblasen;
      L     W#16#2000;
      OW    ;
      T     #t_zeit_Abblasen;
      SET   ;
      SAVE  ;
      CLR   ;
_017: U     BIE;
      )     ;
      SPBNB _018;
      L     #t_zeit_Abblasen;
      T     #t_S5Time_Zeit_Abblasen;
      SET   ;
      SAVE  ;
      CLR   ;
_018: U     BIE;
      )     ;
      L     #t_S5Time_Zeit_Abblasen;
      SV    "SV_RPL_abblasen";
      NOP   0;
      NOP   0;
      NOP   0;
      NOP   0;
NETWORK
TITLE =Handbedienung Vorrichtung abblasen
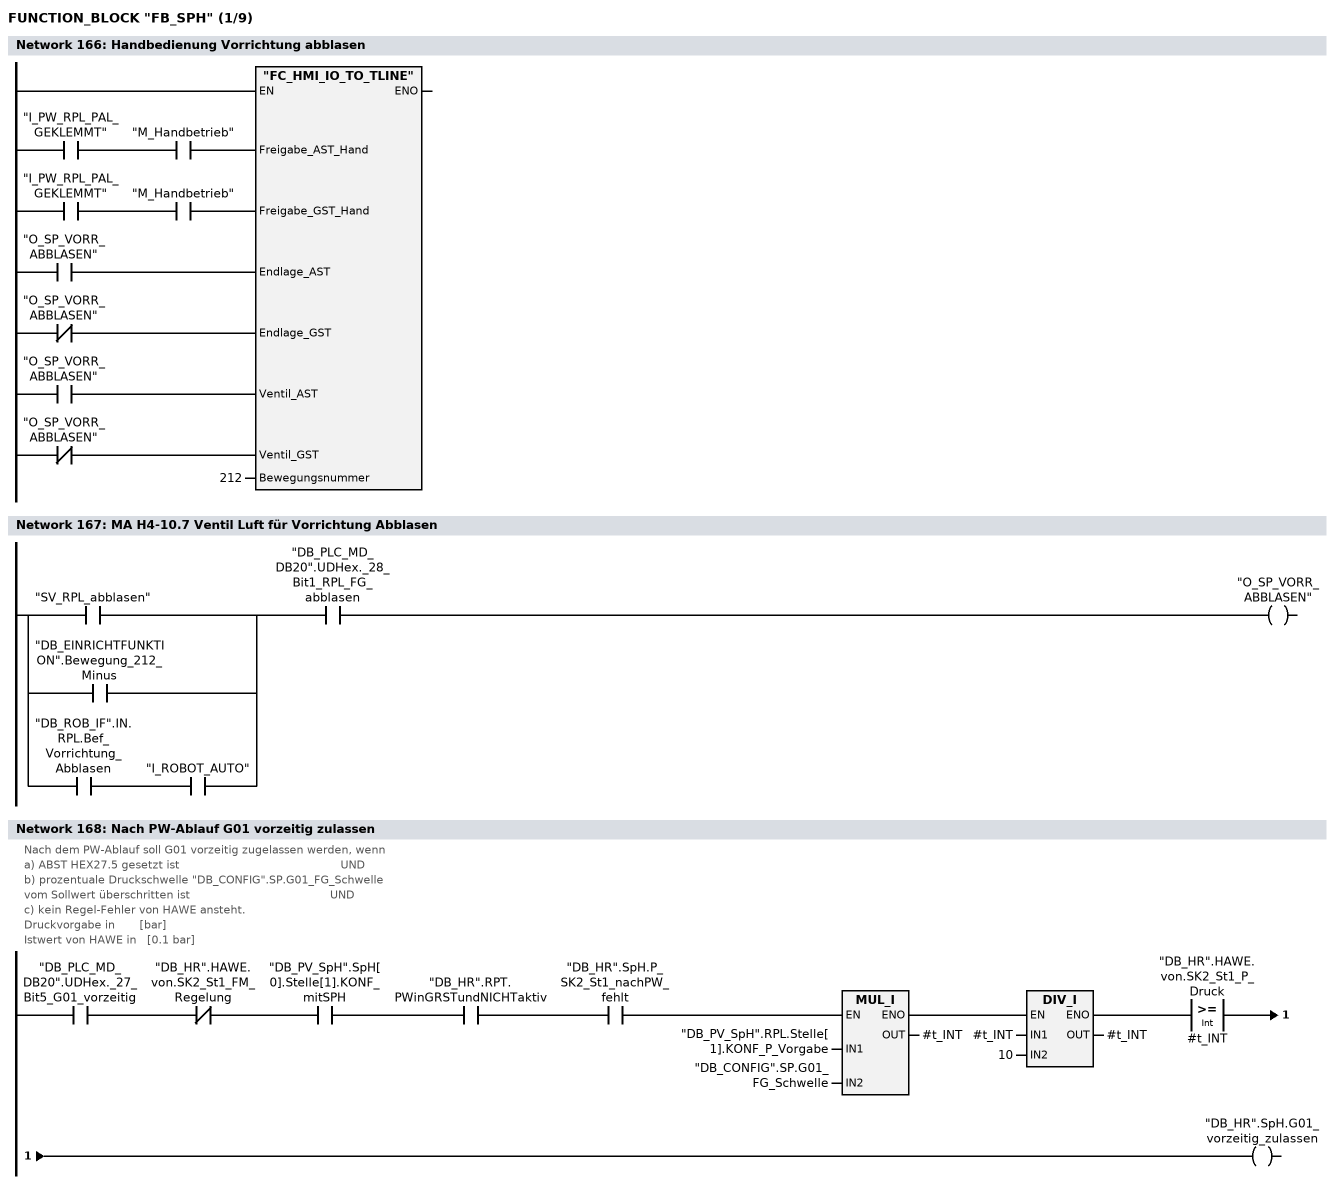

      U     "I_PW_RPL_PAL_GEKLEMMT";
      U     "M_Handbetrieb";
      =     L     18.0;
      BLD   103;
      U     "I_PW_RPL_PAL_GEKLEMMT";
      U     "M_Handbetrieb";
      =     L     18.1;
      BLD   103;
      U     "O_SP_VORR_ABBLASEN";
      =     L     18.2;
      BLD   103;
      UN    "O_SP_VORR_ABBLASEN";
      =     L     18.3;
      BLD   103;
      U     "O_SP_VORR_ABBLASEN";
      =     L     18.4;
      BLD   103;
      UN    "O_SP_VORR_ABBLASEN";
      =     L     18.5;
      BLD   103;
      CALL "FC_HMI_IO_TO_TLINE" (
           Freigabe_AST_Hand        := L     18.0,
           Freigabe_GST_Hand        := L     18.1,
           Endlage_AST              := L     18.2,
           Endlage_GST              := L     18.3,
           Ventil_AST               := L     18.4,
           Ventil_GST               := L     18.5,
           Bewegungsnummer          := 212);
      NOP   0;
NETWORK
TITLE =MA H4-10.7 Ventil Luft für Vorrichtung Abblasen

      U(    ;
      O     "SV_RPL_abblasen";
      O     "DB_EINRICHTFUNKTION".Bewegung_212_Minus;
      O     ;
      U     "DB_ROB_IF".IN.RPL.Bef_Vorrichtung_Abblasen;
      U     "I_ROBOT_AUTO";
      )     ;
      U     "DB_PLC_MD_DB20".UDHex._28_Bit1_RPL_FG_abblasen;
      =     "O_SP_VORR_ABBLASEN";
NETWORK
TITLE =Nach PW-Ablauf G01 vorzeitig zulassen
//Nach dem PW-Ablauf soll G01 vorzeitig zugelassen werden, wenn
//a) ABST HEX27.5 gesetzt ist                                              UND
//b) prozentuale Druckschwelle "DB_CONFIG".SP.G01_FG_Schwelle
//   vom Sollwert überschritten ist                                        UND
//c) kein Regel-Fehler von HAWE ansteht.
//
//Druckvorgabe in       [bar]
//Istwert von HAWE in   [0.1 bar]
      U(    ;
      U(    ;
      U     "DB_PLC_MD_DB20".UDHex._27_Bit5_G01_vorzeitig;
      UN    "DB_HR".HAWE.von.SK2_St1_FM_Regelung;
      U     "DB_PV_SpH".SpH[0].Stelle[1].KONF_mitSPH;
      U     "DB_HR".RPT.PWinGRSTundNICHTaktiv;
      U     "DB_HR".SpH.P_SK2_St1_nachPW_fehlt;
      SPBNB _019;
      L     "DB_PV_SpH".RPL.Stelle[1].KONF_P_Vorgabe;
      L     "DB_CONFIG".SP.G01_FG_Schwelle;
      *I    ;
      T     #t_INT;
      UN    OV;
      SAVE  ;
      CLR   ;
_019: U     BIE;
      )     ;
      SPBNB _01a;
      L     #t_INT;
      L     10;
      /I    ;
      T     #t_INT;
      UN    OV;
      SAVE  ;
      CLR   ;
_01a: U     BIE;
      )     ;
      U(    ;
      L     "DB_HR".HAWE.von.SK2_St1_P_Druck;
      L     #t_INT;
      >=I   ;
      )     ;
      =     "DB_HR".SpH.G01_vorzeitig_zulassen;
NETWORK
TITLE =Vorschub-Sperre SpannHydraulik
//H31=Spannstelle 1    H32=Spannstelle 2    H33=Spannstelle 3    H34=Spannstelle 4
//H31=x (20 <= x <= 240) Druckänderung auf Spannstelle 1
//H31=0                  Ausschalten Drucküberwachung Spannstelle 1
//                       Einschalten mit H31=x oder Palettenwechsel
//H31=-x (0 <= x <= 200) Entspannen Spannstelle 1 (Öffnen)
//                       mit Druck=150 bar und Zeit xx Wert in [100 ms]
